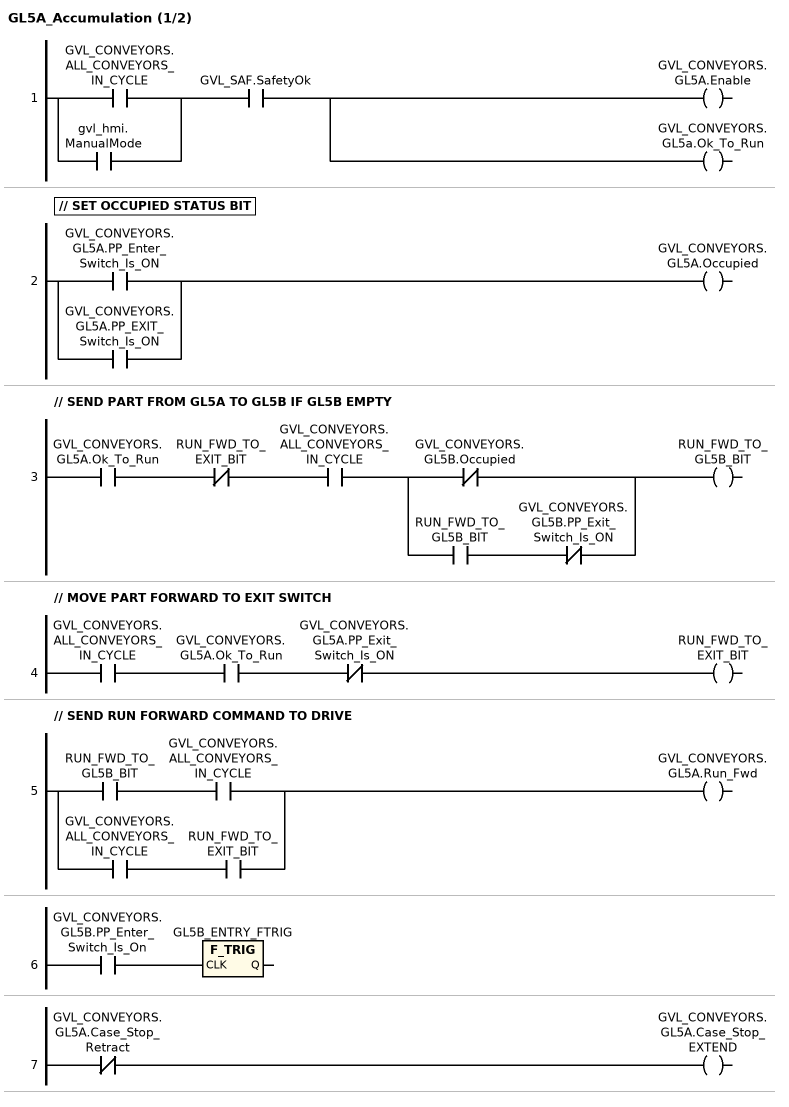
// NETWORK 1
_w1 := (GVL_CONVEYORS.ALL_CONVEYORS_IN_CYCLE OR gvl_hmi.ManualMode) AND GVL_SAF.SafetyOk;
GVL_CONVEYORS.GL5A.Enable := _w1;
GVL_CONVEYORS.GL5a.Ok_To_Run := _w1;

// NETWORK 2
// label: // SET OCCUPIED STATUS BIT
GVL_CONVEYORS.GL5A.Occupied := GVL_CONVEYORS.GL5A.PP_Enter_Switch_Is_ON OR GVL_CONVEYORS.GL5A.PP_EXIT_Switch_Is_ON;

// NETWORK 3: // SEND PART FROM GL5A TO GL5B IF GL5B EMPTY
RUN_FWD_TO_GL5B_BIT := GVL_CONVEYORS.GL5A.Ok_To_Run AND NOT RUN_FWD_TO_EXIT_BIT AND GVL_CONVEYORS.ALL_CONVEYORS_IN_CYCLE AND (NOT GVL_CONVEYORS.GL5B.Occupied OR RUN_FWD_TO_GL5B_BIT AND NOT GVL_CONVEYORS.GL5B.PP_Exit_Switch_Is_ON);

// NETWORK 4: // MOVE PART FORWARD TO EXIT SWITCH
RUN_FWD_TO_EXIT_BIT := GVL_CONVEYORS.ALL_CONVEYORS_IN_CYCLE AND GVL_CONVEYORS.GL5A.Ok_To_Run AND NOT GVL_CONVEYORS.GL5A.PP_Exit_Switch_Is_ON;

// NETWORK 5: // SEND RUN FORWARD COMMAND TO DRIVE
GVL_CONVEYORS.GL5A.Run_Fwd := RUN_FWD_TO_GL5B_BIT AND GVL_CONVEYORS.ALL_CONVEYORS_IN_CYCLE OR GVL_CONVEYORS.ALL_CONVEYORS_IN_CYCLE AND RUN_FWD_TO_EXIT_BIT;

// NETWORK 6
GL5B_ENTRY_FTRIG(CLK := GVL_CONVEYORS.GL5B.PP_Enter_Switch_Is_On); // F_TRIG

// NETWORK 7
GVL_CONVEYORS.GL5A.Case_Stop_EXTEND := NOT GVL_CONVEYORS.GL5A.Case_Stop_Retract;

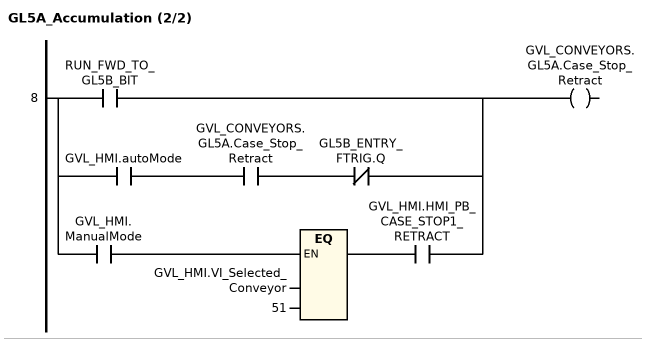
// NETWORK 8
GVL_CONVEYORS.GL5A.Case_Stop_Retract := RUN_FWD_TO_GL5B_BIT OR GVL_HMI.autoMode AND GVL_CONVEYORS.GL5A.Case_Stop_Retract AND NOT GL5B_ENTRY_FTRIG.Q OR (GVL_HMI.ManualMode AND GVL_HMI.VI_Selected_Conveyor = 51) AND GVL_HMI.HMI_PB_CASE_STOP1_RETRACT;

END_PROGRAM

// ---- Machine System/PRGs/Conveyors/GL5B_Accumulation.TcPOU
PROGRAM GL5B_Accumulation
VAR
	
	RUN_FWD_TO_GL2_BIT : BOOL; // GL2 EMPTY SO SEND PART FROM GL5B TO GL2
	RUN_FWD_TO_EXIT_BIT : BOOL; // RUN GL5B FWD TO EXIT SENSOR
	
END_VAR
VAR // added by the converter: edge detectors and wires of the graphical bodies
    _w1 : BOOL;
END_VAR

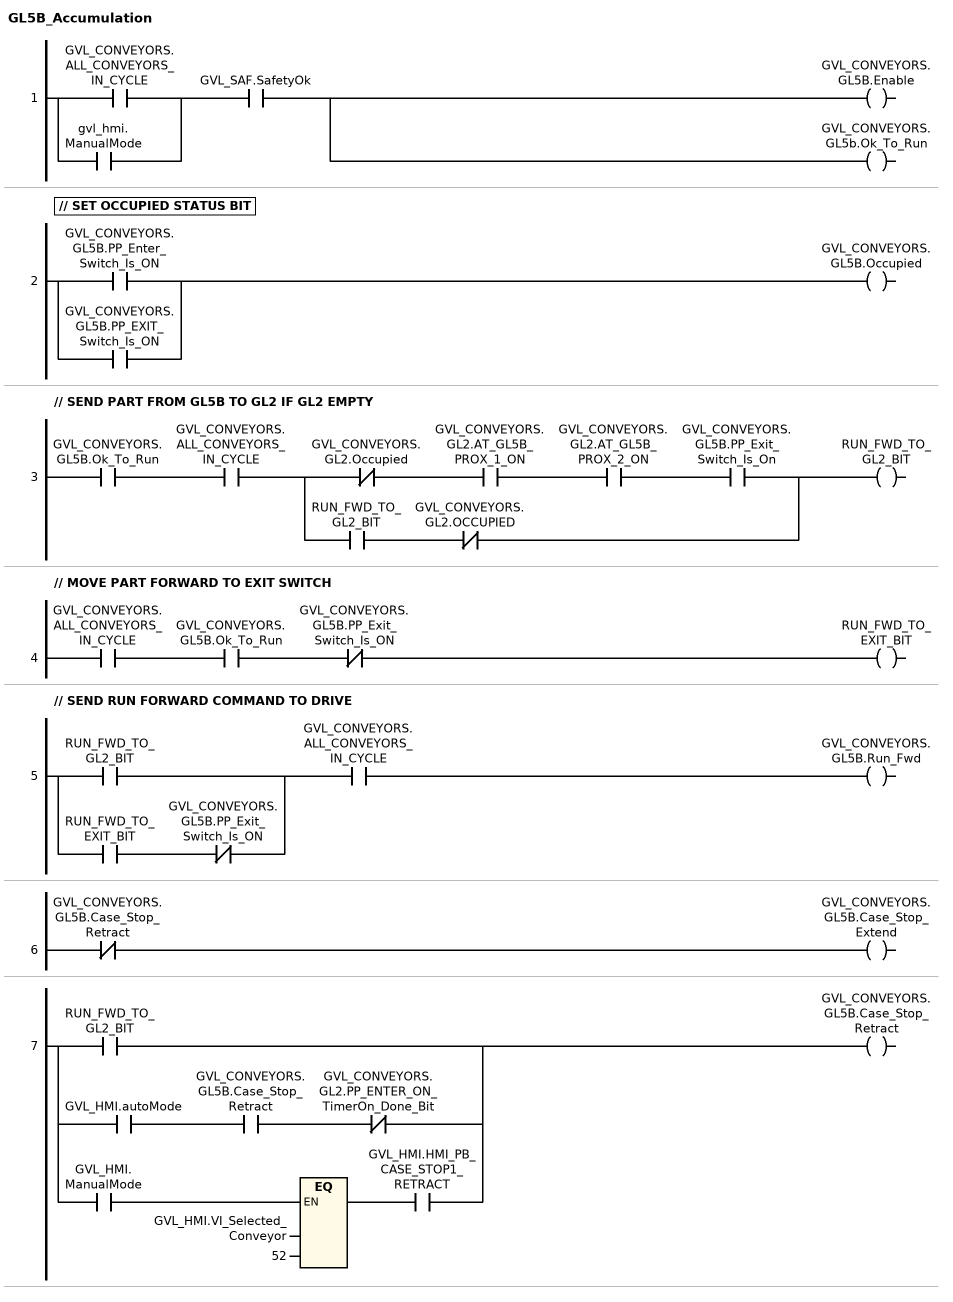
// NETWORK 1
_w1 := (GVL_CONVEYORS.ALL_CONVEYORS_IN_CYCLE OR gvl_hmi.ManualMode) AND GVL_SAF.SafetyOk;
GVL_CONVEYORS.GL5B.Enable := _w1;
GVL_CONVEYORS.GL5b.Ok_To_Run := _w1;

// NETWORK 2
// label: // SET OCCUPIED STATUS BIT
GVL_CONVEYORS.GL5B.Occupied := GVL_CONVEYORS.GL5B.PP_Enter_Switch_Is_ON OR GVL_CONVEYORS.GL5B.PP_EXIT_Switch_Is_ON;

// NETWORK 3: // SEND PART FROM GL5B TO GL2 IF GL2 EMPTY
RUN_FWD_TO_GL2_BIT := GVL_CONVEYORS.GL5B.Ok_To_Run AND GVL_CONVEYORS.ALL_CONVEYORS_IN_CYCLE AND (NOT GVL_CONVEYORS.GL2.Occupied AND GVL_CONVEYORS.GL2.AT_GL5B_PROX_1_ON AND GVL_CONVEYORS.GL2.AT_GL5B_PROX_2_ON AND GVL_CONVEYORS.GL5B.PP_Exit_Switch_Is_On OR RUN_FWD_TO_GL2_BIT AND NOT GVL_CONVEYORS.GL2.OCCUPIED);

// NETWORK 4: // MOVE PART FORWARD TO EXIT SWITCH
RUN_FWD_TO_EXIT_BIT := GVL_CONVEYORS.ALL_CONVEYORS_IN_CYCLE AND GVL_CONVEYORS.GL5B.Ok_To_Run AND NOT GVL_CONVEYORS.GL5B.PP_Exit_Switch_Is_ON;

// NETWORK 5: // SEND RUN FORWARD COMMAND TO DRIVE
GVL_CONVEYORS.GL5B.Run_Fwd := (RUN_FWD_TO_GL2_BIT OR RUN_FWD_TO_EXIT_BIT AND NOT GVL_CONVEYORS.GL5B.PP_Exit_Switch_Is_ON) AND GVL_CONVEYORS.ALL_CONVEYORS_IN_CYCLE;

// NETWORK 6
GVL_CONVEYORS.GL5B.Case_Stop_Extend := NOT GVL_CONVEYORS.GL5B.Case_Stop_Retract;

// NETWORK 7
GVL_CONVEYORS.GL5B.Case_Stop_Retract := RUN_FWD_TO_GL2_BIT OR GVL_HMI.autoMode AND GVL_CONVEYORS.GL5B.Case_Stop_Retract AND NOT GVL_CONVEYORS.GL2.PP_ENTER_ON_TimerOn_Done_Bit OR (GVL_HMI.ManualMode AND GVL_HMI.VI_Selected_Conveyor = 52) AND GVL_HMI.HMI_PB_CASE_STOP1_RETRACT;

END_PROGRAM

// ---- Machine System/PRGs/Conveyors/GL6_Conveyor.TcPOU
PROGRAM GL6_Conveyor
VAR
	GL6_RD: SRoll_Door;
	PASSSED_ROLL_DOOR : BOOL;
	RUN_FWD_BIT_TO_LOAD: BOOL; // RUN FORWARD TO LOAD POSITIONS
	RUN_FWD_BIT_TO_EXIT : BOOL; // RUN FORWARD TO EXIT POSITION AFTER DROP
	JoeBit : BOOL := FALSE;
END_VAR
VAR // added by the converter: edge detectors and wires of the graphical bodies
    _w1 : BOOL;
END_VAR

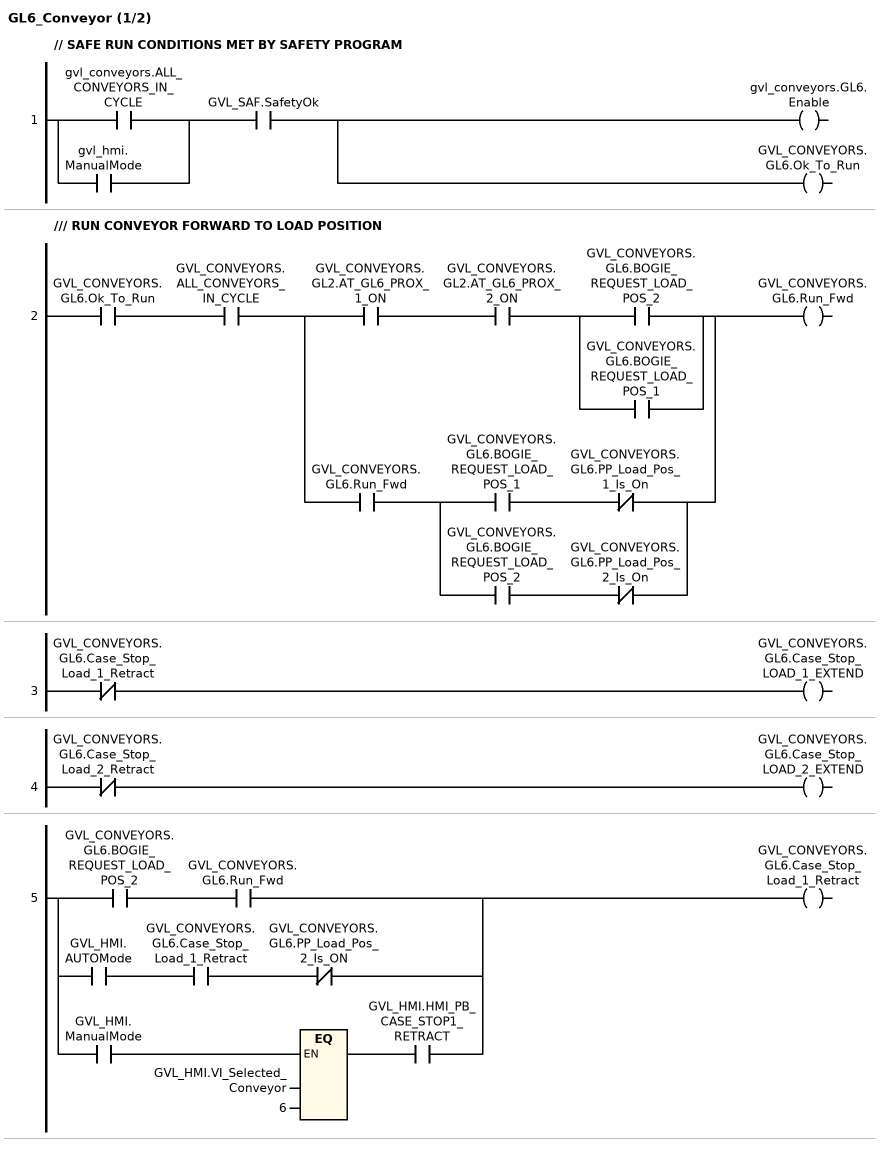
// NETWORK 1: // SAFE RUN CONDITIONS MET BY SAFETY PROGRAM
_w1 := (gvl_conveyors.ALL_CONVEYORS_IN_CYCLE OR gvl_hmi.ManualMode) AND GVL_SAF.SafetyOk;
gvl_conveyors.GL6.Enable := _w1;
GVL_CONVEYORS.GL6.Ok_To_Run := _w1;

// NETWORK 2: /// RUN CONVEYOR FORWARD TO LOAD POSITION
GVL_CONVEYORS.GL6.Run_Fwd := GVL_CONVEYORS.GL6.Ok_To_Run AND GVL_CONVEYORS.ALL_CONVEYORS_IN_CYCLE AND (GVL_CONVEYORS.GL2.AT_GL6_PROX_1_ON AND GVL_CONVEYORS.GL2.AT_GL6_PROX_2_ON AND (GVL_CONVEYORS.GL6.BOGIE_REQUEST_LOAD_POS_2 OR GVL_CONVEYORS.GL6.BOGIE_REQUEST_LOAD_POS_1) OR GVL_CONVEYORS.GL6.Run_Fwd AND (GVL_CONVEYORS.GL6.BOGIE_REQUEST_LOAD_POS_1 AND NOT GVL_CONVEYORS.GL6.PP_Load_Pos_1_Is_On OR GVL_CONVEYORS.GL6.BOGIE_REQUEST_LOAD_POS_2 AND NOT GVL_CONVEYORS.GL6.PP_Load_Pos_2_Is_On));

// NETWORK 3
GVL_CONVEYORS.GL6.Case_Stop_LOAD_1_EXTEND := NOT GVL_CONVEYORS.GL6.Case_Stop_Load_1_Retract;

// NETWORK 4
GVL_CONVEYORS.GL6.Case_Stop_LOAD_2_EXTEND := NOT GVL_CONVEYORS.GL6.Case_Stop_Load_2_Retract;

// NETWORK 5
GVL_CONVEYORS.GL6.Case_Stop_Load_1_Retract := GVL_CONVEYORS.GL6.BOGIE_REQUEST_LOAD_POS_2 AND GVL_CONVEYORS.GL6.Run_Fwd OR GVL_HMI.AUTOMode AND GVL_CONVEYORS.GL6.Case_Stop_Load_1_Retract AND NOT GVL_CONVEYORS.GL6.PP_Load_Pos_2_Is_ON OR (GVL_HMI.ManualMode AND GVL_HMI.VI_Selected_Conveyor = 6) AND GVL_HMI.HMI_PB_CASE_STOP1_RETRACT;

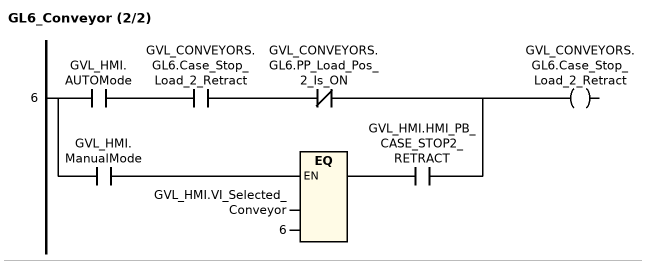
// NETWORK 6
GVL_CONVEYORS.GL6.Case_Stop_Load_2_Retract := GVL_HMI.AUTOMode AND GVL_CONVEYORS.GL6.Case_Stop_Load_2_Retract AND NOT GVL_CONVEYORS.GL6.PP_Load_Pos_2_Is_ON OR (GVL_HMI.ManualMode AND GVL_HMI.VI_Selected_Conveyor = 6) AND GVL_HMI.HMI_PB_CASE_STOP2_RETRACT;

END_PROGRAM

// ---- Machine System/PRGs/Conveyors/GL7_Conveyor.TcPOU
PROGRAM GL7_Conveyor
VAR
	
	RUN_FWD_BIT_TO_EXIT : BOOL; // RUN FORWARD TO EXIT POSITION AFTER DROP
END_VAR
VAR // added by the converter: edge detectors and wires of the graphical bodies
    _w1 : BOOL;
END_VAR

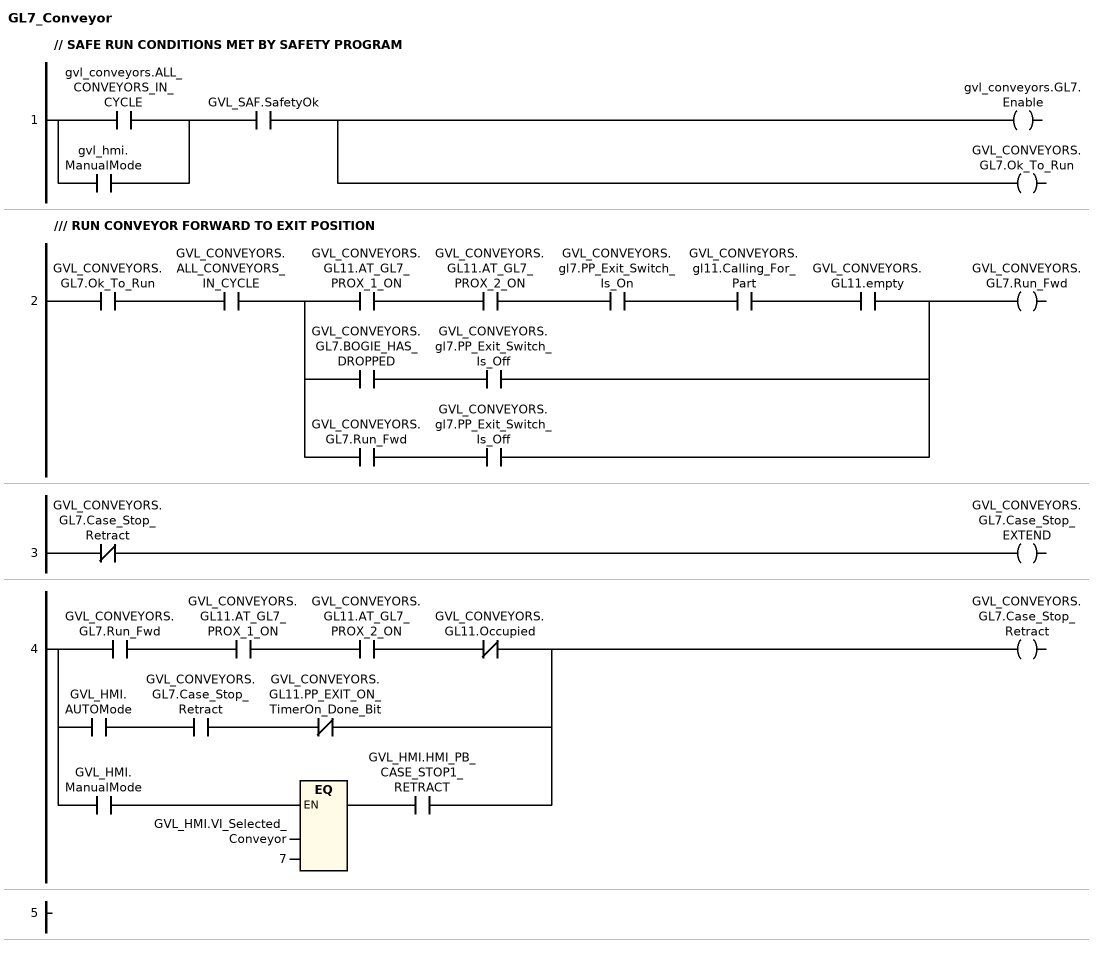
// NETWORK 1: // SAFE RUN CONDITIONS MET BY SAFETY PROGRAM
_w1 := (gvl_conveyors.ALL_CONVEYORS_IN_CYCLE OR gvl_hmi.ManualMode) AND GVL_SAF.SafetyOk;
gvl_conveyors.GL7.Enable := _w1;
GVL_CONVEYORS.GL7.Ok_To_Run := _w1;

// NETWORK 2: /// RUN CONVEYOR FORWARD TO EXIT POSITION
GVL_CONVEYORS.GL7.Run_Fwd := GVL_CONVEYORS.GL7.Ok_To_Run AND GVL_CONVEYORS.ALL_CONVEYORS_IN_CYCLE AND (GVL_CONVEYORS.GL11.AT_GL7_PROX_1_ON AND GVL_CONVEYORS.GL11.AT_GL7_PROX_2_ON AND GVL_CONVEYORS.gl7.PP_Exit_Switch_Is_On AND GVL_CONVEYORS.gl11.Calling_For_Part AND GVL_CONVEYORS.GL11.empty OR GVL_CONVEYORS.GL7.BOGIE_HAS_DROPPED AND GVL_CONVEYORS.gl7.PP_Exit_Switch_Is_Off OR GVL_CONVEYORS.GL7.Run_Fwd AND GVL_CONVEYORS.gl7.PP_Exit_Switch_Is_Off);

// NETWORK 3
GVL_CONVEYORS.GL7.Case_Stop_EXTEND := NOT GVL_CONVEYORS.GL7.Case_Stop_Retract;

// NETWORK 4
GVL_CONVEYORS.GL7.Case_Stop_Retract := GVL_CONVEYORS.GL7.Run_Fwd AND GVL_CONVEYORS.GL11.AT_GL7_PROX_1_ON AND GVL_CONVEYORS.GL11.AT_GL7_PROX_2_ON AND NOT GVL_CONVEYORS.GL11.Occupied OR GVL_HMI.AUTOMode AND GVL_CONVEYORS.GL7.Case_Stop_Retract AND NOT GVL_CONVEYORS.GL11.PP_EXIT_ON_TimerOn_Done_Bit OR (GVL_HMI.ManualMode AND GVL_HMI.VI_Selected_Conveyor = 7) AND GVL_HMI.HMI_PB_CASE_STOP1_RETRACT;

// NETWORK 5

END_PROGRAM

// ---- Machine System/PRGs/Conveyors/GL8_Conveyor.TcPOU
PROGRAM GL8_Conveyor
VAR
	
	GL8_RD: SRoll_Door;
	PASSSED_ROLL_DOOR : BOOL;
	RUN_FWD_BIT_TO_LOAD: BOOL; // RUN FORWARD TO LOAD POSITIONS
	RUN_FWD_BIT_TO_EXIT : BOOL; // RUN FORWARD TO EXIT POSITION AFTER DROP
	
END_VAR
VAR // added by the converter: edge detectors and wires of the graphical bodies
    _w1 : BOOL;
END_VAR

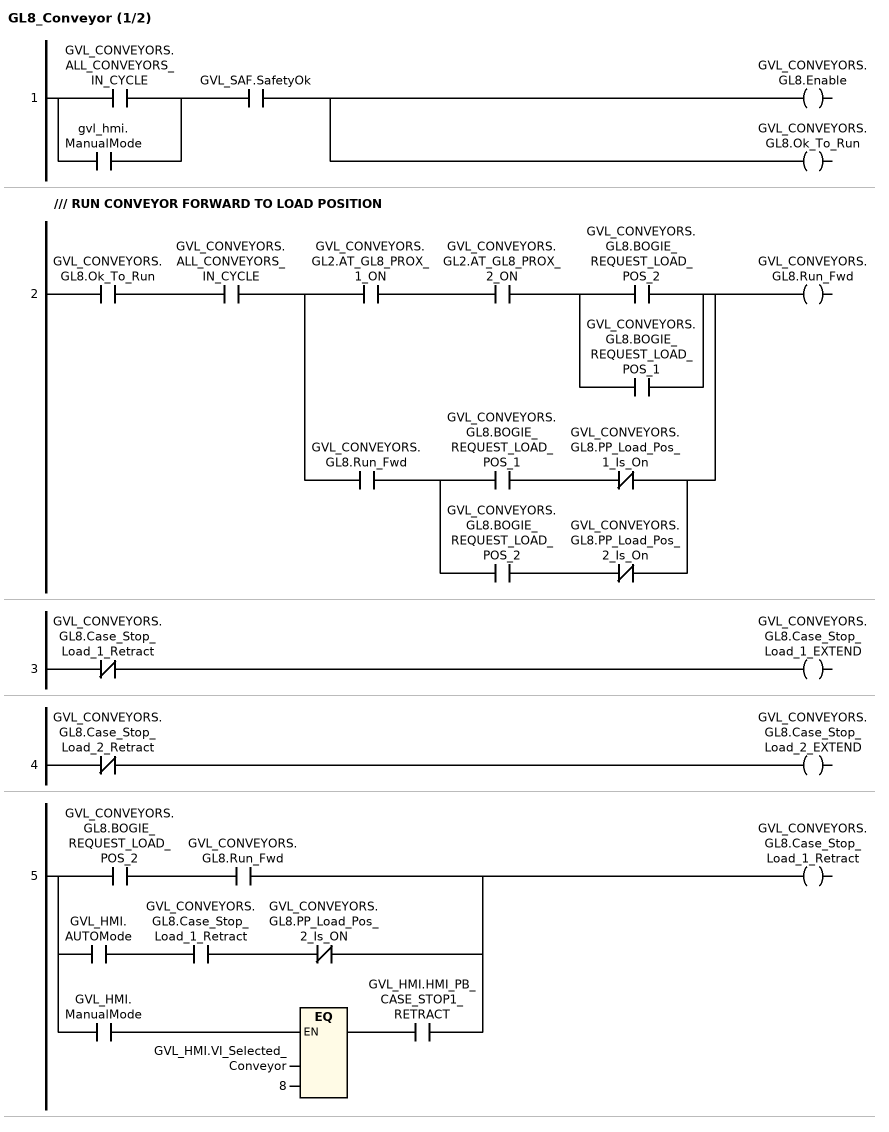
// NETWORK 1
_w1 := (GVL_CONVEYORS.ALL_CONVEYORS_IN_CYCLE OR gvl_hmi.ManualMode) AND GVL_SAF.SafetyOk;
GVL_CONVEYORS.GL8.Enable := _w1;
GVL_CONVEYORS.GL8.Ok_To_Run := _w1;

// NETWORK 2: /// RUN CONVEYOR FORWARD TO LOAD POSITION
GVL_CONVEYORS.GL8.Run_Fwd := GVL_CONVEYORS.GL8.Ok_To_Run AND GVL_CONVEYORS.ALL_CONVEYORS_IN_CYCLE AND (GVL_CONVEYORS.GL2.AT_GL8_PROX_1_ON AND GVL_CONVEYORS.GL2.AT_GL8_PROX_2_ON AND (GVL_CONVEYORS.GL8.BOGIE_REQUEST_LOAD_POS_2 OR GVL_CONVEYORS.GL8.BOGIE_REQUEST_LOAD_POS_1) OR GVL_CONVEYORS.GL8.Run_Fwd AND (GVL_CONVEYORS.GL8.BOGIE_REQUEST_LOAD_POS_1 AND NOT GVL_CONVEYORS.GL8.PP_Load_Pos_1_Is_On OR GVL_CONVEYORS.GL8.BOGIE_REQUEST_LOAD_POS_2 AND NOT GVL_CONVEYORS.GL8.PP_Load_Pos_2_Is_On));

// NETWORK 3
GVL_CONVEYORS.GL8.Case_Stop_Load_1_EXTEND := NOT GVL_CONVEYORS.GL8.Case_Stop_Load_1_Retract;

// NETWORK 4
GVL_CONVEYORS.GL8.Case_Stop_Load_2_EXTEND := NOT GVL_CONVEYORS.GL8.Case_Stop_Load_2_Retract;

// NETWORK 5
GVL_CONVEYORS.GL8.Case_Stop_Load_1_Retract := GVL_CONVEYORS.GL8.BOGIE_REQUEST_LOAD_POS_2 AND GVL_CONVEYORS.GL8.Run_Fwd OR GVL_HMI.AUTOMode AND GVL_CONVEYORS.GL8.Case_Stop_Load_1_Retract AND NOT GVL_CONVEYORS.GL8.PP_Load_Pos_2_Is_ON OR (GVL_HMI.ManualMode AND GVL_HMI.VI_Selected_Conveyor = 8) AND GVL_HMI.HMI_PB_CASE_STOP1_RETRACT;

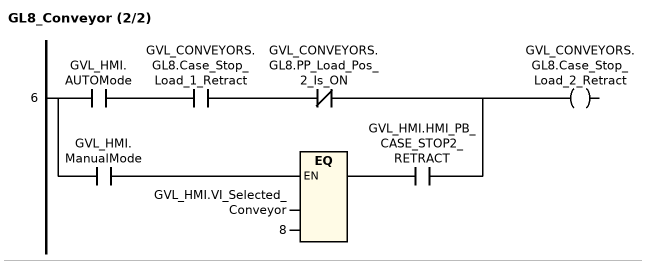
// NETWORK 6
GVL_CONVEYORS.GL8.Case_Stop_Load_2_Retract := GVL_HMI.AUTOMode AND GVL_CONVEYORS.GL8.Case_Stop_Load_1_Retract AND NOT GVL_CONVEYORS.GL8.PP_Load_Pos_2_Is_ON OR (GVL_HMI.ManualMode AND GVL_HMI.VI_Selected_Conveyor = 8) AND GVL_HMI.HMI_PB_CASE_STOP2_RETRACT;

END_PROGRAM

// ---- Machine System/PRGs/Conveyors/GL9_Conveyor.TcPOU
PROGRAM GL9_Conveyor
VAR
	
	RUN_FWD_BIT_TO_EXIT : BOOL; // RUN FORWARD TO EXIT POSITION AFTER DROP
END_VAR
VAR // added by the converter: edge detectors and wires of the graphical bodies
    _w1 : BOOL;
END_VAR

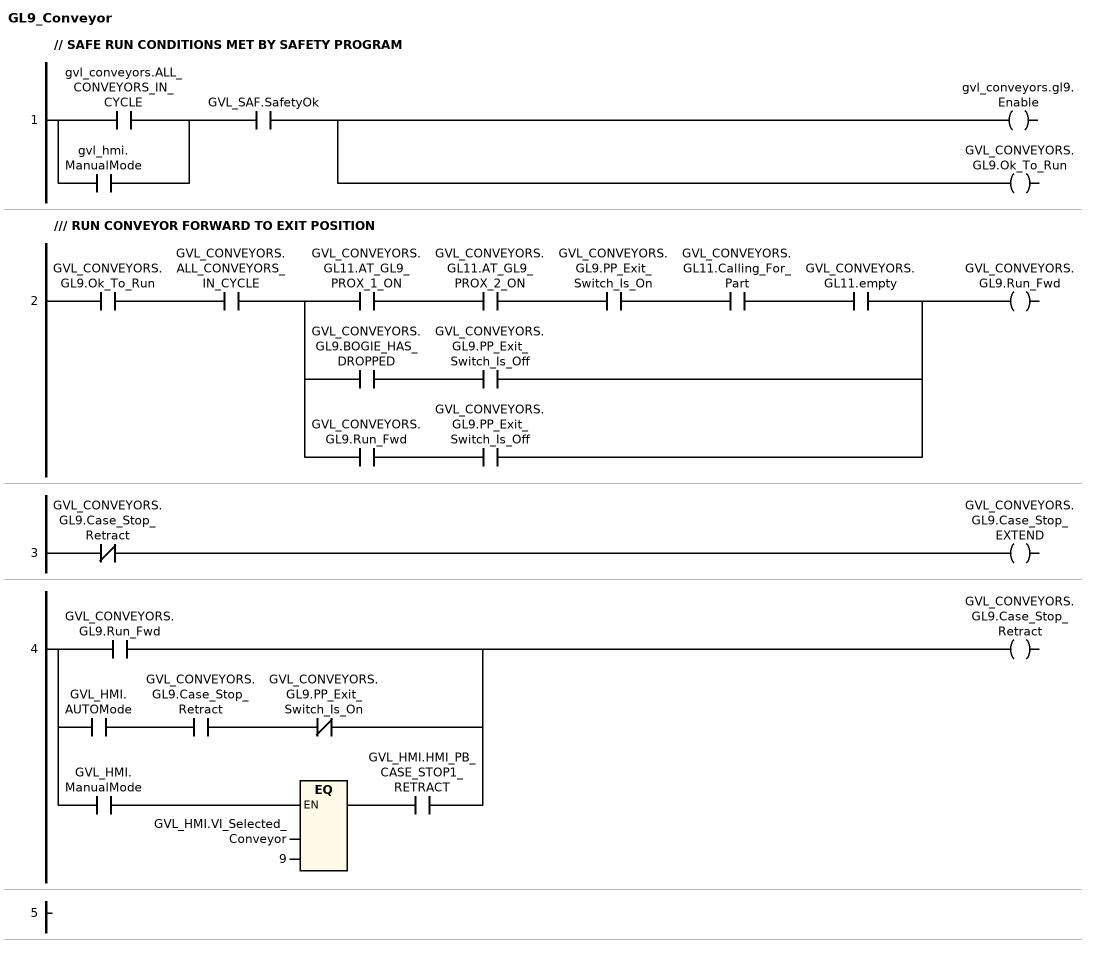
// NETWORK 1: // SAFE RUN CONDITIONS MET BY SAFETY PROGRAM
_w1 := (gvl_conveyors.ALL_CONVEYORS_IN_CYCLE OR gvl_hmi.ManualMode) AND GVL_SAF.SafetyOk;
gvl_conveyors.gl9.Enable := _w1;
GVL_CONVEYORS.GL9.Ok_To_Run := _w1;

// NETWORK 2: /// RUN CONVEYOR FORWARD TO EXIT POSITION
GVL_CONVEYORS.GL9.Run_Fwd := GVL_CONVEYORS.GL9.Ok_To_Run AND GVL_CONVEYORS.ALL_CONVEYORS_IN_CYCLE AND (GVL_CONVEYORS.GL11.AT_GL9_PROX_1_ON AND GVL_CONVEYORS.GL11.AT_GL9_PROX_2_ON AND GVL_CONVEYORS.GL9.PP_Exit_Switch_Is_On AND GVL_CONVEYORS.GL11.Calling_For_Part AND GVL_CONVEYORS.GL11.empty OR GVL_CONVEYORS.GL9.BOGIE_HAS_DROPPED AND GVL_CONVEYORS.GL9.PP_Exit_Switch_Is_Off OR GVL_CONVEYORS.GL9.Run_Fwd AND GVL_CONVEYORS.GL9.PP_Exit_Switch_Is_Off);

// NETWORK 3
GVL_CONVEYORS.GL9.Case_Stop_EXTEND := NOT GVL_CONVEYORS.GL9.Case_Stop_Retract;

// NETWORK 4
GVL_CONVEYORS.GL9.Case_Stop_Retract := GVL_CONVEYORS.GL9.Run_Fwd OR GVL_HMI.AUTOMode AND GVL_CONVEYORS.GL9.Case_Stop_Retract AND NOT GVL_CONVEYORS.GL9.PP_Exit_Switch_Is_On OR (GVL_HMI.ManualMode AND GVL_HMI.VI_Selected_Conveyor = 9) AND GVL_HMI.HMI_PB_CASE_STOP1_RETRACT;

// NETWORK 5

END_PROGRAM

// ---- Machine System/PRGs/Rib Machine/Guarding_Safety.TcPOU
PROGRAM Guarding_Safety
VAR
END_VAR

// NETWORK 1

END_PROGRAM

// ---- Machine System/PRGs/Rib Machine/Input_Buffering_RB.TcPOU
PROGRAM Input_Buffering_RB
VAR PERSISTENT
	
	StackerPartPresentTon: TON;
	StackerPinExtendedTon: TON;
	StackerPinRetractedTon: TON;
	IndexerPartPresentTon: TON;
    SawExtendedTon: TON;
	SawRetractedTon: TON;
	SawClampExtendedTon: TON;
	SawClampRetractedTon: TON;
	SawClampOpenTon: TON;
	SawClampClosedTon: TON;
	TransferClampOpenTon: TON;
	TransferClampClosedTon: TON;
	TransferClampExtdTon: TON;
	TransferClampRetdTon: TON;
	TransferExtdTon: TON;
	TransferRetdTon: TON;
	RibHoistUpTon: TON;
	RibHoistDownTon: TON;
	EjectExtendedTon: TON;
	EjectRetractedTon: TON;
	AirPressureSwitchTon: TON;
	IndexerHomeTon: TON;
	
END_VAR

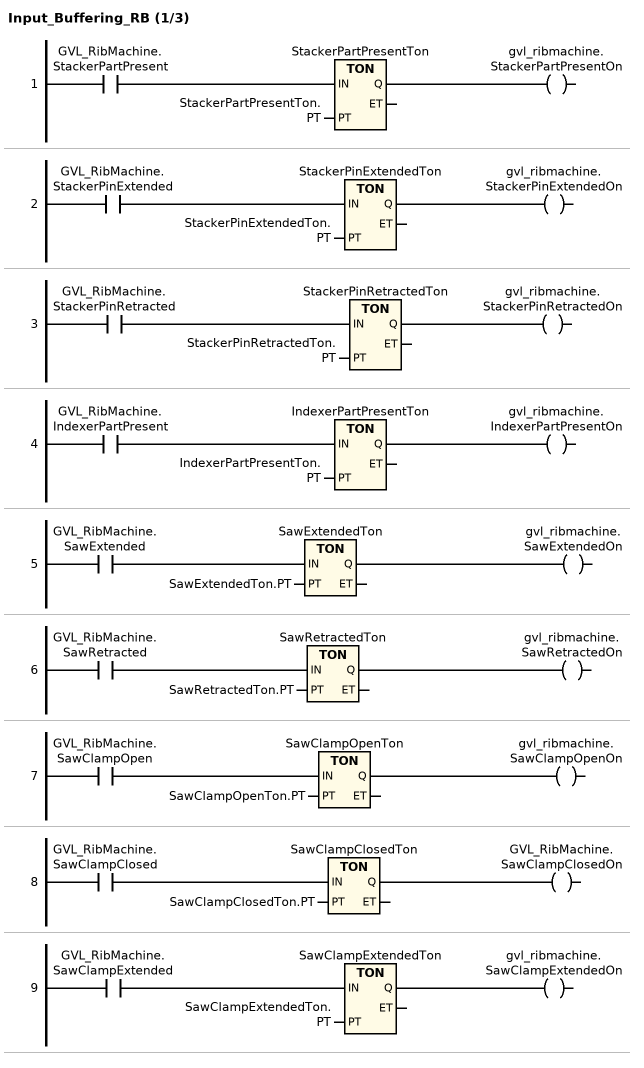
// NETWORK 1
StackerPartPresentTon(IN := GVL_RibMachine.StackerPartPresent, PT := StackerPartPresentTon.PT); // TON
gvl_ribmachine.StackerPartPresentOn := StackerPartPresentTon.Q;

// NETWORK 2
StackerPinExtendedTon(IN := GVL_RibMachine.StackerPinExtended, PT := StackerPinExtendedTon.PT); // TON
gvl_ribmachine.StackerPinExtendedOn := StackerPinExtendedTon.Q;

// NETWORK 3
StackerPinRetractedTon(IN := GVL_RibMachine.StackerPinRetracted, PT := StackerPinRetractedTon.PT); // TON
gvl_ribmachine.StackerPinRetractedOn := StackerPinRetractedTon.Q;

// NETWORK 4
IndexerPartPresentTon(IN := GVL_RibMachine.IndexerPartPresent, PT := IndexerPartPresentTon.PT); // TON
gvl_ribmachine.IndexerPartPresentOn := IndexerPartPresentTon.Q;

// NETWORK 5
SawExtendedTon(IN := GVL_RibMachine.SawExtended, PT := SawExtendedTon.PT); // TON
gvl_ribmachine.SawExtendedOn := SawExtendedTon.Q;

// NETWORK 6
SawRetractedTon(IN := GVL_RibMachine.SawRetracted, PT := SawRetractedTon.PT); // TON
gvl_ribmachine.SawRetractedOn := SawRetractedTon.Q;

// NETWORK 7
SawClampOpenTon(IN := GVL_RibMachine.SawClampOpen, PT := SawClampOpenTon.PT); // TON
gvl_ribmachine.SawClampOpenOn := SawClampOpenTon.Q;

// NETWORK 8
SawClampClosedTon(IN := GVL_RibMachine.SawClampClosed, PT := SawClampClosedTon.PT); // TON
GVL_RibMachine.SawClampClosedOn := SawClampClosedTon.Q;

// NETWORK 9
SawClampExtendedTon(IN := GVL_RibMachine.SawClampExtended, PT := SawClampExtendedTon.PT); // TON
gvl_ribmachine.SawClampExtendedOn := SawClampExtendedTon.Q;

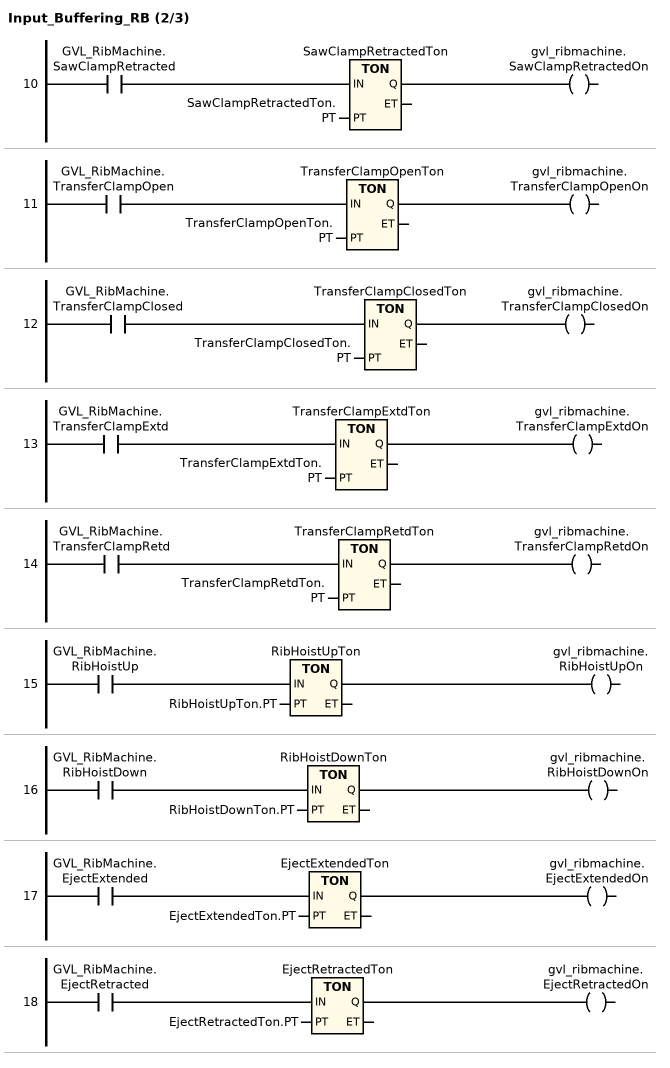
// NETWORK 10
SawClampRetractedTon(IN := GVL_RibMachine.SawClampRetracted, PT := SawClampRetractedTon.PT); // TON
gvl_ribmachine.SawClampRetractedOn := SawClampRetractedTon.Q;

// NETWORK 11
TransferClampOpenTon(IN := GVL_RibMachine.TransferClampOpen, PT := TransferClampOpenTon.PT); // TON
gvl_ribmachine.TransferClampOpenOn := TransferClampOpenTon.Q;

// NETWORK 12
TransferClampClosedTon(IN := GVL_RibMachine.TransferClampClosed, PT := TransferClampClosedTon.PT); // TON
gvl_ribmachine.TransferClampClosedOn := TransferClampClosedTon.Q;

// NETWORK 13
TransferClampExtdTon(IN := GVL_RibMachine.TransferClampExtd, PT := TransferClampExtdTon.PT); // TON
gvl_ribmachine.TransferClampExtdOn := TransferClampExtdTon.Q;

// NETWORK 14
TransferClampRetdTon(IN := GVL_RibMachine.TransferClampRetd, PT := TransferClampRetdTon.PT); // TON
gvl_ribmachine.TransferClampRetdOn := TransferClampRetdTon.Q;

// NETWORK 15
RibHoistUpTon(IN := GVL_RibMachine.RibHoistUp, PT := RibHoistUpTon.PT); // TON
gvl_ribmachine.RibHoistUpOn := RibHoistUpTon.Q;

// NETWORK 16
RibHoistDownTon(IN := GVL_RibMachine.RibHoistDown, PT := RibHoistDownTon.PT); // TON
gvl_ribmachine.RibHoistDownOn := RibHoistDownTon.Q;

// NETWORK 17
EjectExtendedTon(IN := GVL_RibMachine.EjectExtended, PT := EjectExtendedTon.PT); // TON
gvl_ribmachine.EjectExtendedOn := EjectExtendedTon.Q;

// NETWORK 18
EjectRetractedTon(IN := GVL_RibMachine.EjectRetracted, PT := EjectRetractedTon.PT); // TON
gvl_ribmachine.EjectRetractedOn := EjectRetractedTon.Q;

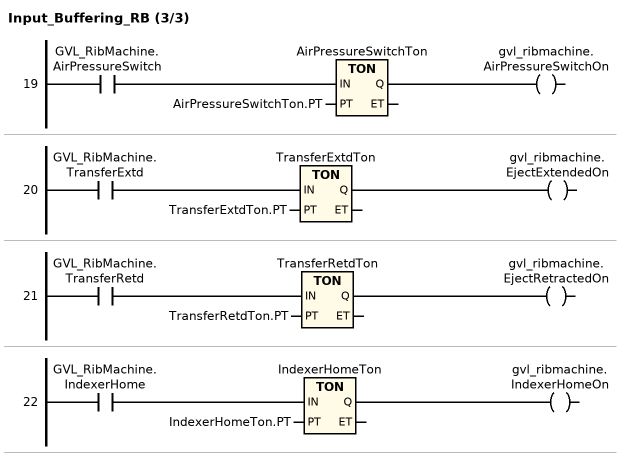
// NETWORK 19
AirPressureSwitchTon(IN := GVL_RibMachine.AirPressureSwitch, PT := AirPressureSwitchTon.PT); // TON
gvl_ribmachine.AirPressureSwitchOn := AirPressureSwitchTon.Q;

// NETWORK 20
TransferExtdTon(IN := GVL_RibMachine.TransferExtd, PT := TransferExtdTon.PT); // TON
gvl_ribmachine.EjectExtendedOn := TransferExtdTon.Q;

// NETWORK 21
TransferRetdTon(IN := GVL_RibMachine.TransferRetd, PT := TransferRetdTon.PT); // TON
gvl_ribmachine.EjectRetractedOn := TransferRetdTon.Q;

// NETWORK 22
IndexerHomeTon(IN := GVL_RibMachine.IndexerHome, PT := IndexerHomeTon.PT); // TON
gvl_ribmachine.IndexerHomeOn := IndexerHomeTon.Q;

END_PROGRAM

// ---- Machine System/PRGs/START_STOP.TcPOU
PROGRAM START_STOP
VAR
	START_TIMER : TON;
	START_TIMER_ELAPSED: TIME;
	START_TIMER_DONE : BOOL; 
	ALARM_HORN AT %Q* : BOOL; // CONVEYOR STARTING WARNING SIGNAL
	ALL_CONVEYORS_START_PB  AT %I*:  BOOL; // TIE THIS TO THE START COMMAND FROM HMI OR BUTTON
	ALL_CONVEYORS_STOP_PB  AT %I*: BOOL; // TIE THIS TO THE STOP COMMAND FROM HMI OR BUTTON
	START_PB_LT AT %Q*: BOOL; // START PB LIGHT
	STOP_PB_LT AT %Q*: BOOL; // STOP PB LIGHT
	KIRK_BIT: BOOL;
	HMI_CONVEYOR_START: BOOL; // START SIGNAL FROM HMI
	
END_VAR

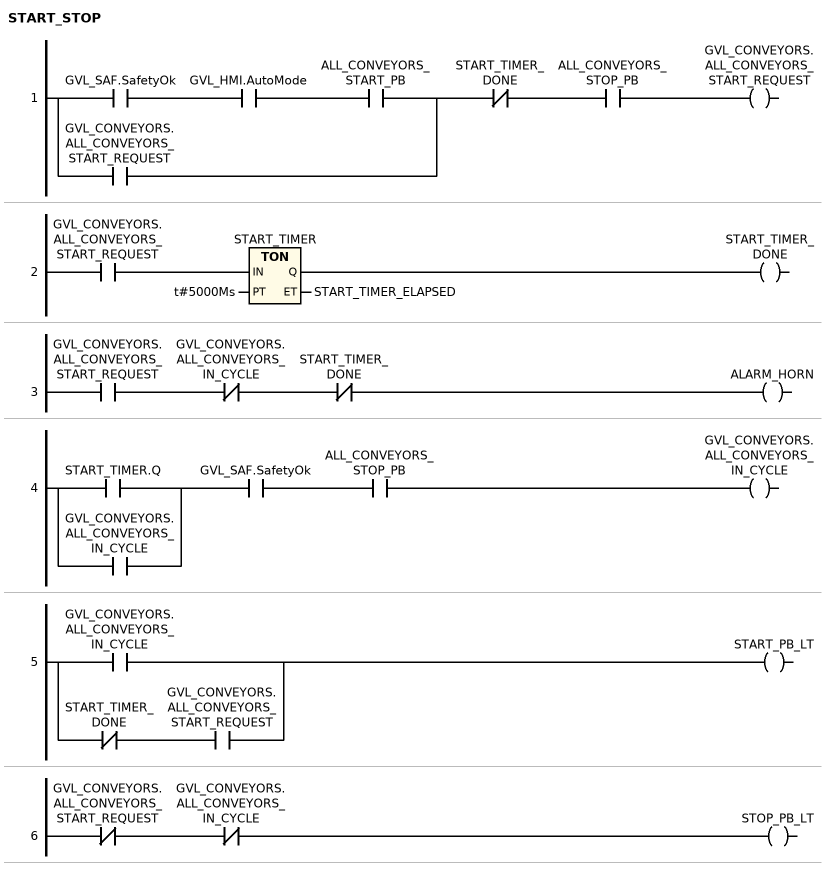
// NETWORK 1
GVL_CONVEYORS.ALL_CONVEYORS_START_REQUEST := (GVL_SAF.SafetyOk AND GVL_HMI.AutoMode AND ALL_CONVEYORS_START_PB OR GVL_CONVEYORS.ALL_CONVEYORS_START_REQUEST) AND NOT START_TIMER_DONE AND ALL_CONVEYORS_STOP_PB;

// NETWORK 2
START_TIMER(IN := GVL_CONVEYORS.ALL_CONVEYORS_START_REQUEST, PT := t#5000Ms, ET => START_TIMER_ELAPSED); // TON
START_TIMER_DONE := START_TIMER.Q;

// NETWORK 3
ALARM_HORN := GVL_CONVEYORS.ALL_CONVEYORS_START_REQUEST AND NOT GVL_CONVEYORS.ALL_CONVEYORS_IN_CYCLE AND NOT START_TIMER_DONE;

// NETWORK 4
GVL_CONVEYORS.ALL_CONVEYORS_IN_CYCLE := (START_TIMER.Q OR GVL_CONVEYORS.ALL_CONVEYORS_IN_CYCLE) AND GVL_SAF.SafetyOk AND ALL_CONVEYORS_STOP_PB;

// NETWORK 5
START_PB_LT := GVL_CONVEYORS.ALL_CONVEYORS_IN_CYCLE OR NOT START_TIMER_DONE AND GVL_CONVEYORS.ALL_CONVEYORS_START_REQUEST;

// NETWORK 6
STOP_PB_LT := NOT GVL_CONVEYORS.ALL_CONVEYORS_START_REQUEST AND NOT GVL_CONVEYORS.ALL_CONVEYORS_IN_CYCLE;

END_PROGRAM

// ---- Machine System/PRGs/Rib Machine/Index_and_Measure.TcPOU
PROGRAM Index_and_Measure
VAR
	RequestedRibLength:REAL; // Length in inches needed for ribs to cut
	MinRibLength: DINT; // Minimnm length of leftover that can still be used.
	MaxRibLength: DINT; // Longest rib lenght
	NumOfRibs:INT; // Quantity of tibs needed for next part
	RibRequest:BOOL; // Ribs needed for next part.
	RemainingLength:DINT; // Left over length of rib after cut
	PPI:REAL; // Pulses Per Inch from encoder
	CutLength: REAL; // Rib length to cut in encoder pulses 
	KerfWidth : REAL; // Width of saw blade in encoder pulses
	TotalCutLength : REAL; // Cut length requested plus kerf width of saw blade
	RibReadyToCut: BOOL; // Rib is in position to begin cutting
	HMI_PB_ManualJogFwd:BOOL; // HMI manual jog forward
	HMI_PB_ManualJogRev: bool; // HMI manual jog reverse
	IndexFwd: BOOL; // Clear path signal to go forward direction
	IndexRev: BOOL; // Clear path signal to go reverse direction
	OpenTransferClampRequest: BOOL;
	CloseTransferClampRequest: BOOL;
END_VAR

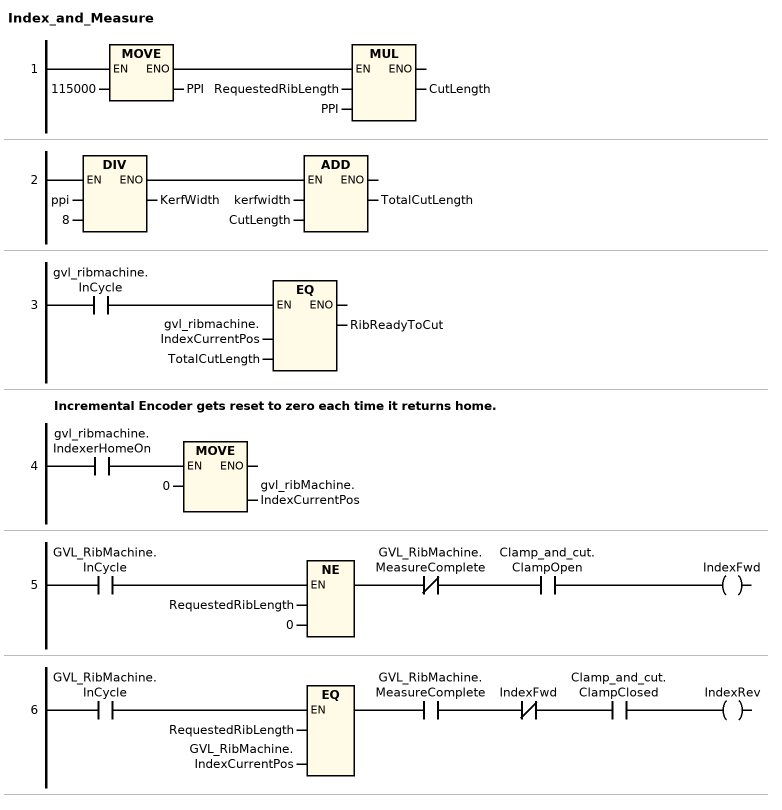
// NETWORK 1
PPI := 115000;
CutLength := RequestedRibLength * PPI;

// NETWORK 2
KerfWidth := ppi / 8;
TotalCutLength := kerfwidth + CutLength;

// NETWORK 3
IF gvl_ribmachine.InCycle THEN RibReadyToCut := gvl_ribmachine.IndexCurrentPos = TotalCutLength; END_IF

// NETWORK 4: Incremental Encoder gets reset to zero each time it returns home.
IF gvl_ribmachine.IndexerHomeOn THEN gvl_ribMachine.IndexCurrentPos := 0; END_IF

// NETWORK 5
IndexFwd := (GVL_RibMachine.InCycle AND RequestedRibLength <> 0) AND NOT GVL_RibMachine.MeasureComplete AND Clamp_and_cut.ClampOpen;

// NETWORK 6
IndexRev := (GVL_RibMachine.InCycle AND RequestedRibLength = GVL_RibMachine.IndexCurrentPos) AND GVL_RibMachine.MeasureComplete AND NOT IndexFwd AND Clamp_and_cut.ClampClosed;

END_PROGRAM

// ---- Machine System/PRGs/Rib Machine/Clamp_and_cut.TcPOU
PROGRAM Clamp_and_cut
VAR
	
	
	SawHome: BOOL; //Indexer is retracted to HOME switch
	SawTraversing: BOOL; // Saw is cycling through cutting
	SawDwellTimer: ton; // Dwell timer to wait for saw to spool up to speed
	SawExtended: BOOL; // Saw slide is fully extended
	ClampOpen: BOOL; // Saw clamp is open to receive part
	ClampClosed: BOOL; // Saw clamp is closed on to the part
	SawMotorRunning: BOOL; // Saw blade is spinning and motor not faulted
	CloseClampRequest: BOOL; // Logic bit to close saw clamp
	OpenClampRequest: BOOL; // Logic bit to open saw clamp
	SawDwellTimerElapsed: TIME; // Elapsed time of dwell timer
	SawDwellDoneBit: BOOL; // Dwell timer done bit
	StartSawRequest: BOOL; // Logic bit to start saw motor
	TraverseDwellTimer: ton; // Dwell timer to wait for traverse motor to spool up to speed
	TraverseDwellTimerElapsed: TIME; // Elapsed time of dwell timer
	TraverseDwellDoneBit: BOOL; // Dwell timer done bit
	DustCollectStartRequest: BOOL; // Logic bit to start dust collector
	
END_VAR
VAR // added by the converter: edge detectors and wires of the graphical bodies
    _rt1, _rt2, _rt3 : R_TRIG;
    _w1 : BOOL;
END_VAR

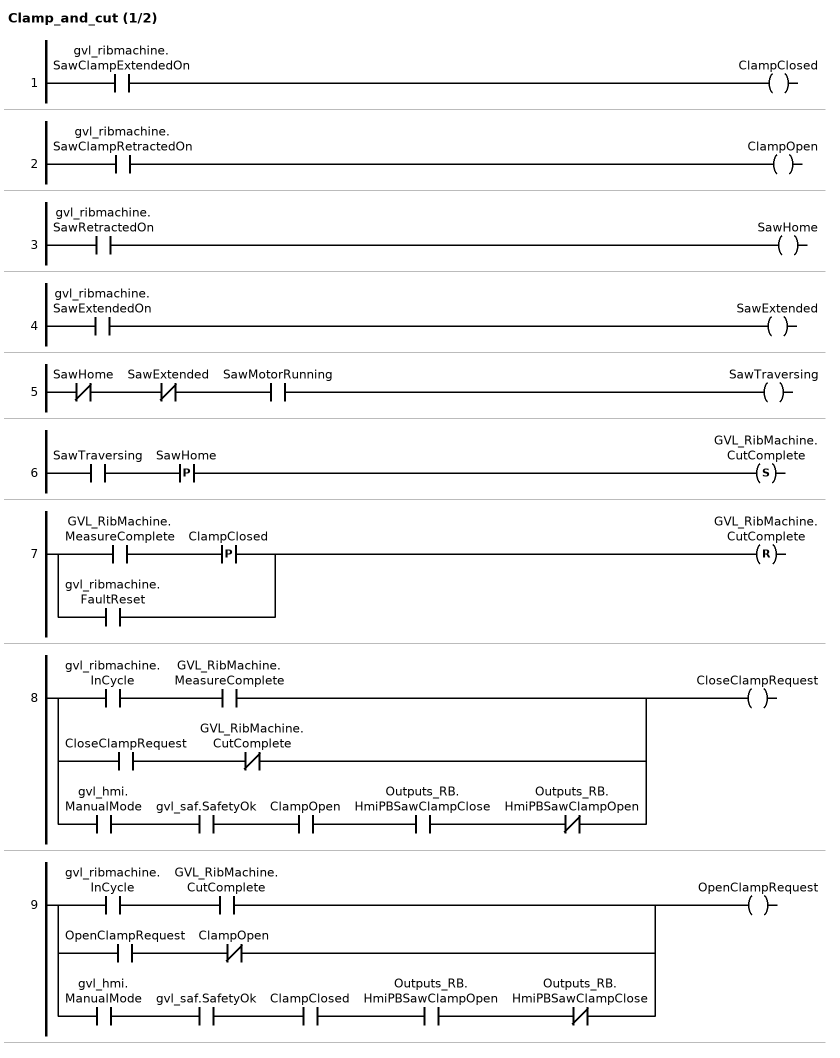
// NETWORK 1
ClampClosed := gvl_ribmachine.SawClampExtendedOn;

// NETWORK 2
ClampOpen := gvl_ribmachine.SawClampRetractedOn;

// NETWORK 3
SawHome := gvl_ribmachine.SawRetractedOn;

// NETWORK 4
SawExtended := gvl_ribmachine.SawExtendedOn;

// NETWORK 5
SawTraversing := NOT SawHome AND NOT SawExtended AND SawMotorRunning;

// NETWORK 6
_rt1(CLK := SawHome);
GVL_RibMachine.CutComplete S= SawTraversing AND _rt1.Q;

// NETWORK 7
_rt2(CLK := ClampClosed);
GVL_RibMachine.CutComplete R= GVL_RibMachine.MeasureComplete AND _rt2.Q OR gvl_ribmachine.FaultReset;

// NETWORK 8
CloseClampRequest := gvl_ribmachine.InCycle AND GVL_RibMachine.MeasureComplete OR CloseClampRequest AND NOT GVL_RibMachine.CutComplete OR gvl_hmi.ManualMode AND gvl_saf.SafetyOk AND ClampOpen AND Outputs_RB.HmiPBSawClampClose AND NOT Outputs_RB.HmiPBSawClampOpen;

// NETWORK 9
OpenClampRequest := gvl_ribmachine.InCycle AND GVL_RibMachine.CutComplete OR OpenClampRequest AND NOT ClampOpen OR gvl_hmi.ManualMode AND gvl_saf.SafetyOk AND ClampClosed AND Outputs_RB.HmiPBSawClampOpen AND NOT Outputs_RB.HmiPBSawClampClose;

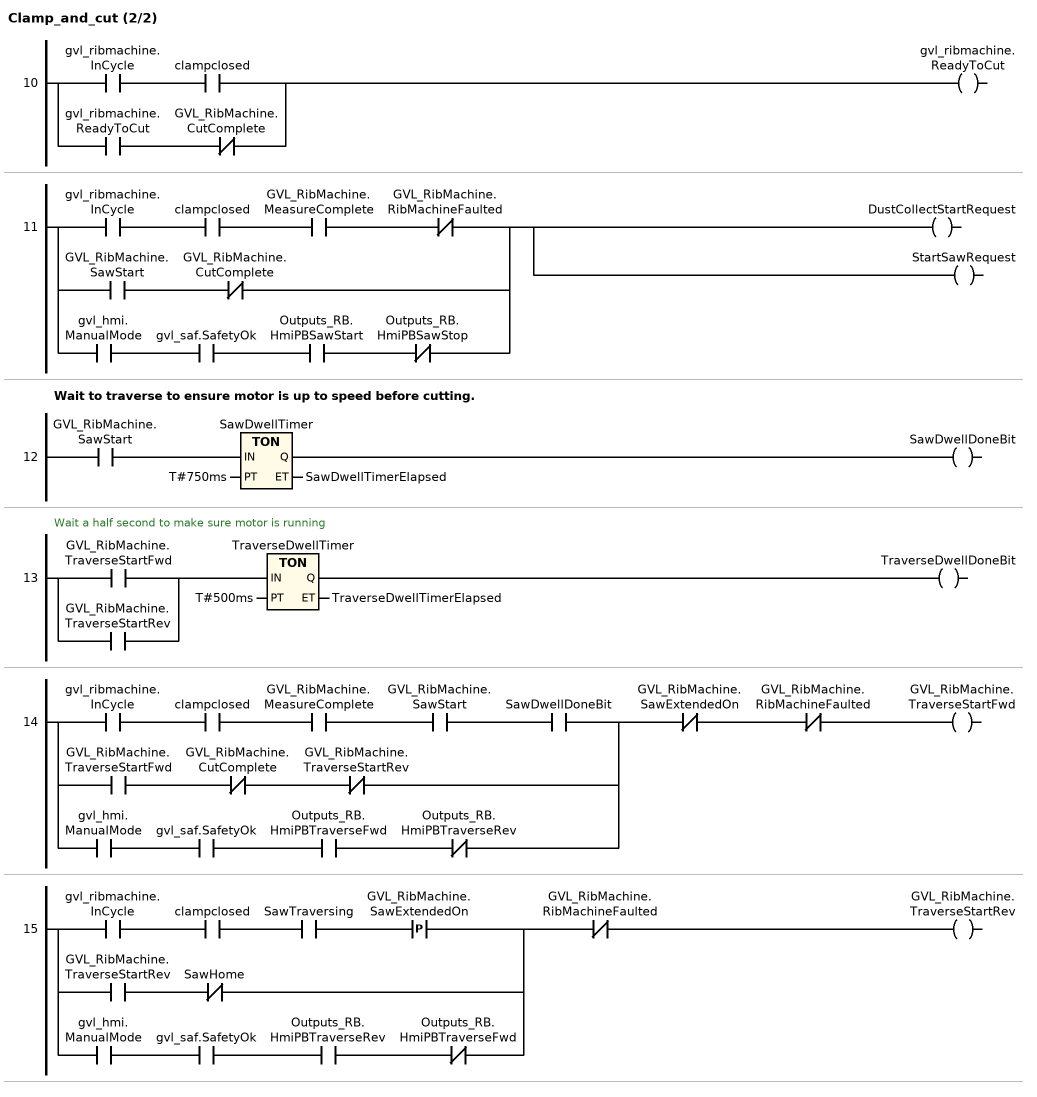
// NETWORK 10
gvl_ribmachine.ReadyToCut := gvl_ribmachine.InCycle AND clampclosed OR gvl_ribmachine.ReadyToCut AND NOT GVL_RibMachine.CutComplete;

// NETWORK 11
_w1 := gvl_ribmachine.InCycle AND clampclosed AND GVL_RibMachine.MeasureComplete AND NOT GVL_RibMachine.RibMachineFaulted OR GVL_RibMachine.SawStart AND NOT GVL_RibMachine.CutComplete OR gvl_hmi.ManualMode AND gvl_saf.SafetyOk AND Outputs_RB.HmiPBSawStart AND NOT Outputs_RB.HmiPBSawStop;
DustCollectStartRequest := _w1;
StartSawRequest := _w1;

// NETWORK 12: Wait to traverse to ensure motor is up to speed before cutting.
SawDwellTimer(IN := GVL_RibMachine.SawStart, PT := T#750ms, ET => SawDwellTimerElapsed); // TON
SawDwellDoneBit := SawDwellTimer.Q;

// NETWORK 13
// Wait a half second to make sure motor is running
TraverseDwellTimer(
    IN := GVL_RibMachine.TraverseStartFwd OR GVL_RibMachine.TraverseStartRev,
    PT := T#500ms,
    ET => TraverseDwellTimerElapsed); // TON
TraverseDwellDoneBit := TraverseDwellTimer.Q;

// NETWORK 14
GVL_RibMachine.TraverseStartFwd := (gvl_ribmachine.InCycle AND clampclosed AND GVL_RibMachine.MeasureComplete AND GVL_RibMachine.SawStart AND SawDwellDoneBit OR GVL_RibMachine.TraverseStartFwd AND NOT GVL_RibMachine.CutComplete AND NOT GVL_RibMachine.TraverseStartRev OR gvl_hmi.ManualMode AND gvl_saf.SafetyOk AND Outputs_RB.HmiPBTraverseFwd AND NOT Outputs_RB.HmiPBTraverseRev) AND NOT GVL_RibMachine.SawExtendedOn AND NOT GVL_RibMachine.RibMachineFaulted;

// NETWORK 15
_rt3(CLK := GVL_RibMachine.SawExtendedOn);
GVL_RibMachine.TraverseStartRev := (gvl_ribmachine.InCycle AND clampclosed AND SawTraversing AND _rt3.Q OR GVL_RibMachine.TraverseStartRev AND NOT SawHome OR gvl_hmi.ManualMode AND gvl_saf.SafetyOk AND Outputs_RB.HmiPBTraverseRev AND NOT Outputs_RB.HmiPBTraverseFwd) AND NOT GVL_RibMachine.RibMachineFaulted;

END_PROGRAM

// ---- Machine System/PRGs/Rib Machine/Outputs_RB.TcPOU
PROGRAM Outputs_RB
VAR
	HmiPBDoorRequest: BOOL;
	HmiPBIndexFwd: BOOL;
	HmiPBIndexRev: BOOL;
	HmiPBDustCollect: BOOL;
	HmiPBSawStart: BOOL;
	HmiPBSawStop: BOOL;
	HmiPBTraverseFwd: BOOL;
	HmiPBTraverseRev: BOOL;
	HmiPBLiftRaise: BOOL;
	HmiPBLiftLower: BOOL;
	HmiPBTransferFwd: BOOL;
	HmiPBTransferRev: BOOL;
	HmiPBTransferClampOpen: BOOL;
	HmiPBTransferClampClose: BOOL;
	HmiPBTransferClampFwd: BOOL;
	HmiPBTransferClampRev: BOOL;
	HmiPBSawClampClose: BOOL;
	HmiPBSawClampOpen: BOOL;
	HmiPBSawClampFwd: BOOL;
	HmiPBSawClampRev: BOOL;
	HmiPBPinsRaise: BOOL;
	HmiPBPinsLower: BOOL;
	
	
	
	
END_VAR

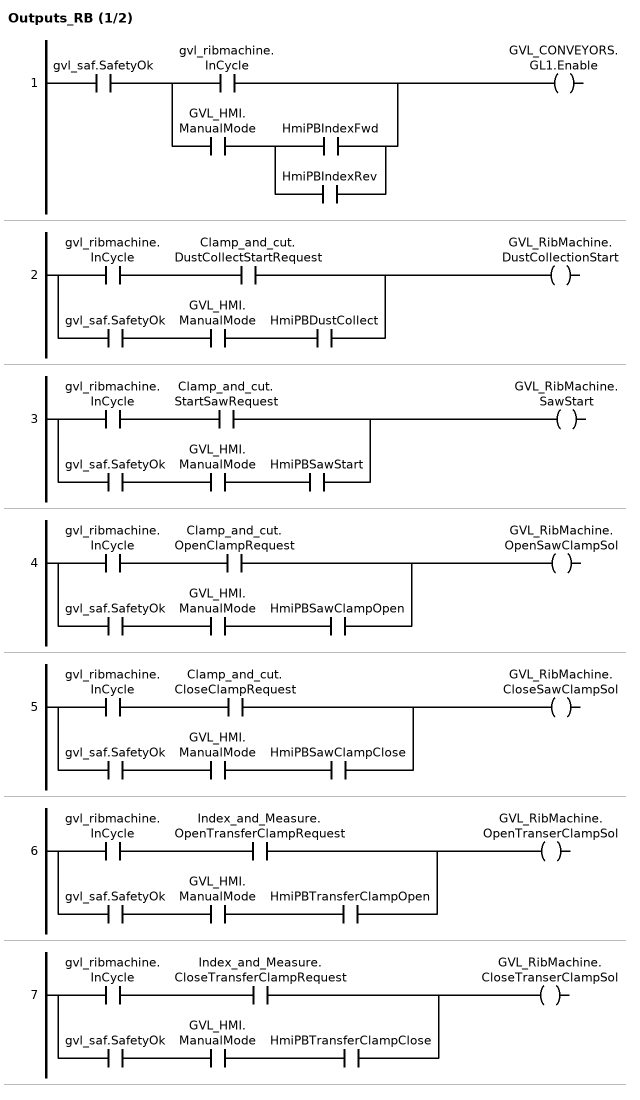
// NETWORK 1
GVL_CONVEYORS.GL1.Enable := gvl_saf.SafetyOk AND (gvl_ribmachine.InCycle OR GVL_HMI.ManualMode AND (HmiPBIndexFwd OR HmiPBIndexRev));

// NETWORK 2
GVL_RibMachine.DustCollectionStart := gvl_ribmachine.InCycle AND Clamp_and_cut.DustCollectStartRequest OR gvl_saf.SafetyOk AND GVL_HMI.ManualMode AND HmiPBDustCollect;

// NETWORK 3
GVL_RibMachine.SawStart := gvl_ribmachine.InCycle AND Clamp_and_cut.StartSawRequest OR gvl_saf.SafetyOk AND GVL_HMI.ManualMode AND HmiPBSawStart;

// NETWORK 4
GVL_RibMachine.OpenSawClampSol := gvl_ribmachine.InCycle AND Clamp_and_cut.OpenClampRequest OR gvl_saf.SafetyOk AND GVL_HMI.ManualMode AND HmiPBSawClampOpen;

// NETWORK 5
GVL_RibMachine.CloseSawClampSol := gvl_ribmachine.InCycle AND Clamp_and_cut.CloseClampRequest OR gvl_saf.SafetyOk AND GVL_HMI.ManualMode AND HmiPBSawClampClose;

// NETWORK 6
GVL_RibMachine.OpenTranserClampSol := gvl_ribmachine.InCycle AND Index_and_Measure.OpenTransferClampRequest OR gvl_saf.SafetyOk AND GVL_HMI.ManualMode AND HmiPBTransferClampOpen;

// NETWORK 7
GVL_RibMachine.CloseTranserClampSol := gvl_ribmachine.InCycle AND Index_and_Measure.CloseTransferClampRequest OR gvl_saf.SafetyOk AND GVL_HMI.ManualMode AND HmiPBTransferClampClose;

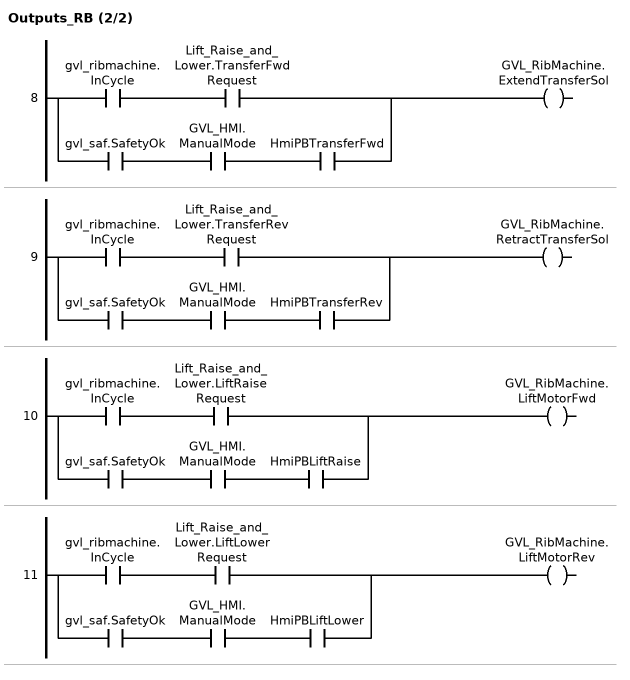
// NETWORK 8
GVL_RibMachine.ExtendTransferSol := gvl_ribmachine.InCycle AND Lift_Raise_and_Lower.TransferFwdRequest OR gvl_saf.SafetyOk AND GVL_HMI.ManualMode AND HmiPBTransferFwd;

// NETWORK 9
GVL_RibMachine.RetractTransferSol := gvl_ribmachine.InCycle AND Lift_Raise_and_Lower.TransferRevRequest OR gvl_saf.SafetyOk AND GVL_HMI.ManualMode AND HmiPBTransferRev;

// NETWORK 10
GVL_RibMachine.LiftMotorFwd := gvl_ribmachine.InCycle AND Lift_Raise_and_Lower.LiftRaiseRequest OR gvl_saf.SafetyOk AND GVL_HMI.ManualMode AND HmiPBLiftRaise;

// NETWORK 11
GVL_RibMachine.LiftMotorRev := gvl_ribmachine.InCycle AND Lift_Raise_and_Lower.LiftLowerRequest OR gvl_saf.SafetyOk AND GVL_HMI.ManualMode AND HmiPBLiftLower;

END_PROGRAM

// ---- Machine System/PRGs/Rib Machine/Lift_Raise_and_Lower.TcPOU
PROGRAM Lift_Raise_and_Lower
VAR
	LiftRaiseRequest: BOOL; // Logic bit to request transfer move forward towards lift bed.
	LiftLowerRequest: BOOL; // Logic bit to request transfer move reverse towards home switch
	ReadyToRaise:BOOL; // Logic bit to indicate ready to lift
	ReadyToLower:BOOL; // Logic bit to indicate ready to lower
	OpenTransferClampRequest:BOOL; // Logic bit to request transfer clamp open
	CloseTransferClampRequest:BOOL; // Logic bit to request transfer clamp close
	TransferFwdRequest: BOOL; // Logic bit to request transfer move forward towards lift bed.
	TransferRevRequest: BOOL; // Logic bit to request transfer move reverse towards home switch
	RibsReadyForPickup:BOOL; // Hoist is up and ribs have been cut to lenght, waiting for gripper to acknowledge pick up
	
END_VAR

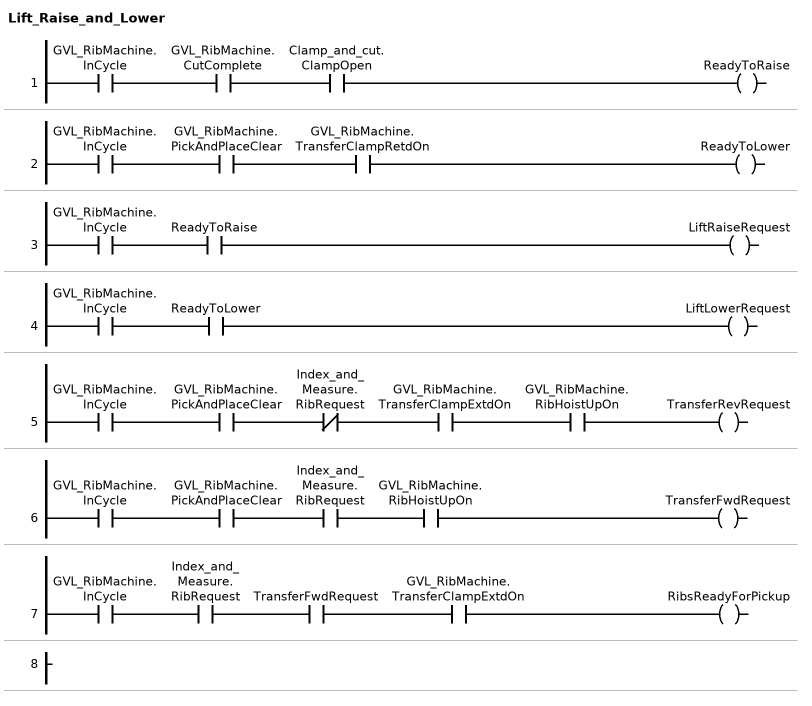
// NETWORK 1
ReadyToRaise := GVL_RibMachine.InCycle AND GVL_RibMachine.CutComplete AND Clamp_and_cut.ClampOpen;

// NETWORK 2
ReadyToLower := GVL_RibMachine.InCycle AND GVL_RibMachine.PickAndPlaceClear AND GVL_RibMachine.TransferClampRetdOn;

// NETWORK 3
LiftRaiseRequest := GVL_RibMachine.InCycle AND ReadyToRaise;

// NETWORK 4
LiftLowerRequest := GVL_RibMachine.InCycle AND ReadyToLower;

// NETWORK 5
TransferRevRequest := GVL_RibMachine.InCycle AND GVL_RibMachine.PickAndPlaceClear AND NOT Index_and_Measure.RibRequest AND GVL_RibMachine.TransferClampExtdOn AND GVL_RibMachine.RibHoistUpOn;

// NETWORK 6
TransferFwdRequest := GVL_RibMachine.InCycle AND GVL_RibMachine.PickAndPlaceClear AND Index_and_Measure.RibRequest AND GVL_RibMachine.RibHoistUpOn;

// NETWORK 7
RibsReadyForPickup := GVL_RibMachine.InCycle AND Index_and_Measure.RibRequest AND TransferFwdRequest AND GVL_RibMachine.TransferClampExtdOn;

// NETWORK 8

END_PROGRAM

// ---- Machine System/PRGs/Rib Machine/Fault_Logic.TcPOU
PROGRAM Fault_Logic
VAR
	
	ScrapBinFullWarning: BOOL;
	RibHopperEmptyFault: BOOL;
	RibHopperNearEmptyWarning: BOOL;
	RibMeasureFault: BOOL;
	LowAirPresFault: BOOL;
	GuardOpenFault: BOOL;
	MotorFault: BOOL;
	JamFault: BOOL;
	AirPresTon : TON;
	AirPresElapsed: TIME;
	
	
	
END_VAR

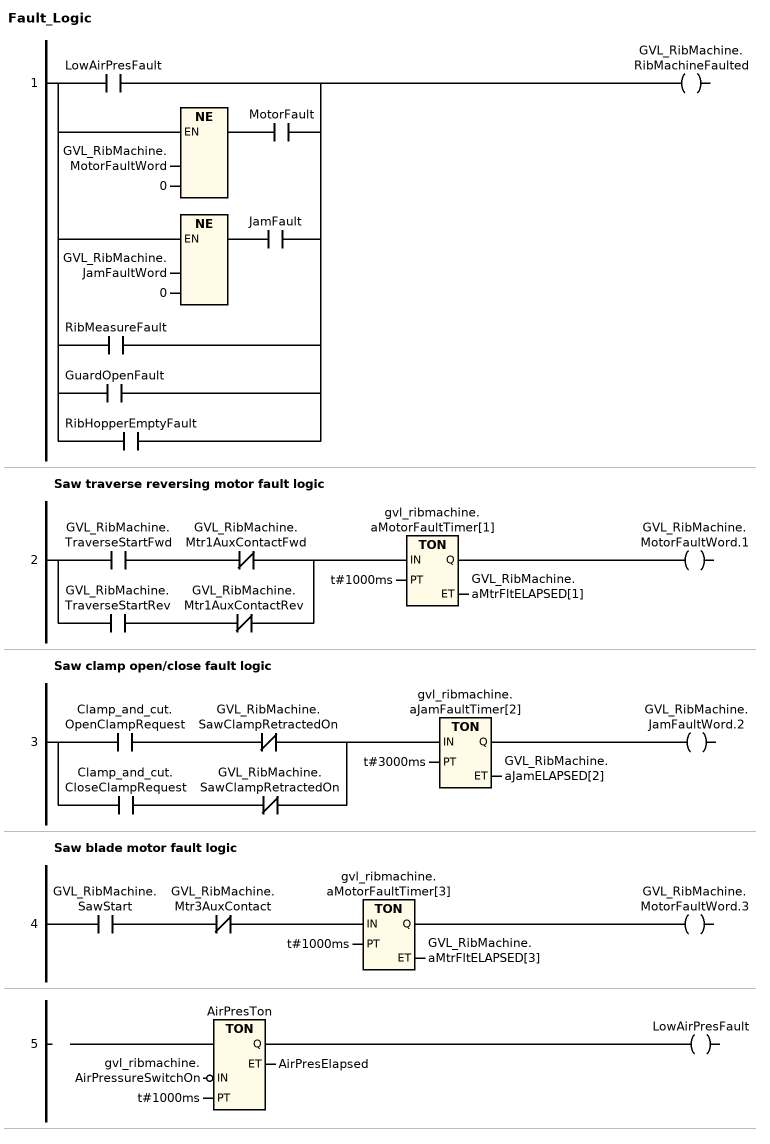
// NETWORK 1
GVL_RibMachine.RibMachineFaulted := LowAirPresFault OR GVL_RibMachine.MotorFaultWord <> 0 AND MotorFault OR GVL_RibMachine.JamFaultWord <> 0 AND JamFault OR RibMeasureFault OR GuardOpenFault OR RibHopperEmptyFault;

// NETWORK 2: Saw traverse reversing motor fault logic
gvl_ribmachine.aMotorFaultTimer[1](
    IN := GVL_RibMachine.TraverseStartFwd AND NOT GVL_RibMachine.Mtr1AuxContactFwd OR GVL_RibMachine.TraverseStartRev AND NOT GVL_RibMachine.Mtr1AuxContactRev,
    PT := t#1000ms,
    ET => GVL_RibMachine.aMtrFltELAPSED[1]); // TON
GVL_RibMachine.MotorFaultWord.1 := gvl_ribmachine.aMotorFaultTimer[1].Q;

// NETWORK 3: Saw clamp open/close fault logic
gvl_ribmachine.aJamFaultTimer[2](
    IN := Clamp_and_cut.OpenClampRequest AND NOT GVL_RibMachine.SawClampRetractedOn OR Clamp_and_cut.CloseClampRequest AND NOT GVL_RibMachine.SawClampRetractedOn,
    PT := t#3000ms,
    ET => GVL_RibMachine.aJamELAPSED[2]); // TON
GVL_RibMachine.JamFaultWord.2 := gvl_ribmachine.aJamFaultTimer[2].Q;

// NETWORK 4: Saw blade motor fault logic
gvl_ribmachine.aMotorFaultTimer[3](
    IN := GVL_RibMachine.SawStart AND NOT GVL_RibMachine.Mtr3AuxContact,
    PT := t#1000ms,
    ET => GVL_RibMachine.aMtrFltELAPSED[3]); // TON
GVL_RibMachine.MotorFaultWord.3 := gvl_ribmachine.aMotorFaultTimer[3].Q;

// NETWORK 5
AirPresTon(IN := NOT gvl_ribmachine.AirPressureSwitchOn, PT := t#1000ms, ET => AirPresElapsed); // TON
LowAirPresFault := AirPresTon.Q;

END_PROGRAM

// ---- Machine System/PRGs/Rib Machine/Interlocks_to_Main_Line.TcPOU
PROGRAM Interlocks_to_Main_Line
VAR
	RibMachineReady: BOOL;
	
	
	
END_VAR

// NETWORK 1

END_PROGRAM

// ---- Machine System/PRGs/ALARM AND STATUS/SYSTEM.TcPOU
PROGRAM SYSTEM
VAR
	fbGetCurTaskIdx  : GETCURTASKINDEX; // PlcTaskSystemInfo for Cycle time
	
	
END_VAR

fbGetCurTaskIdx();
GVL.CycleTime := _TaskInfo[fbGetCurTaskIdx.index].CycleTime/10000;

GVL.GetLocalSystemTimeFB(
	sNetID:= , 
	bEnable:= TRUE, 
	dwCycle:= 1, 
	dwOpt:= , 
	tTimeout:= , 
	bValid=> , 
	systemTime=> , 
	tzID=> );
	
GVL.SystemDateTime := SYSTEMTIME_TO_STRING(GVL.GetLocalSystemTimeFB.systemTime);

GVL.SystemDate := MID(STR:=GVL.SystemDateTime , LEN:=10 , POS:=1 );
GVL.SystemTime := MID(STR:=GVL.SystemDateTime , LEN:=8 , POS:=12 );

END_PROGRAM

// ---- CNC HMI/P_GFunctionMonitor_2.TcPOU
PROGRAM P_GFunctionMonitor_2
VAR
	bReadGcode: BOOL;
	fbADSRead: ADSREADEX;
	GBuffer: ARRAY[1..39]OF WORD;
	nPathPrep: WORD;
	nPlane: WORD;
	nCutterComp: WORD;
	nDeselectDiamProg: WORD;
	nZeroOffset: WORD;
	nContMode: WORD;
	nMeasureMode: WORD;
	nDeselectSpline: WORD;
	nDeselectCornerRed: WORD;
	//toString
		sPathPrep: STRING;
		sPlane: STRING;
		sCutterComp: STRING;
		sDeselectDiamProg: STRING;
		sZeroOffset: STRING;
		sContMode: STRING;
		sMeasureMode: STRING;
		sDeselectSpline: STRING;
		sDeselectCornerRed: STRING;
	fbUpdate: TON;
	sLocalAmsNet 	: STRING; 
	getAmsNet : FB_GetLocalAmsNetId;
	bLocalAmsNet : BOOL;
	
	sGCodeOut : string;
END_VAR

//Read active G code
IF sLocalAmsNet ='' THEN
	bLocalAmsNet := TRUE;
ELSE
	blocalamsNet := FALSE;
END_IF
getAmsNet(bExecute:=bLocalAmsNet, tTimeOut:=DEFAULT_ADS_TIMEOUT,AddrString => sLocalAmsNet);

IF Global_HMI.PLCSelectedChannel = 1 THEN //set this to the selected channel and duplicate for as many channels as necessary
	bReadGcode := TRUE;
	ELSE breadgcode := FALSE;
END_IF

fbUpdate.PT := T#1S;
IF bReadGcode THEN
	fbUpdate.IN := TRUE;
ELSE
	fbUpdate.IN := FALSE;
END_IF

IF fbUpdate.Q THEN
	fbADSRead(
	NETID:=sLocalAmsNet, 
	PORT:=553, 
	IDXGRP:=16#120102, //120102 for ch2 active g code {120101 for ch1}
	IDXOFFS:=16#3C, 
	LEN:=SIZEOF(GBuffer), 
	DESTADDR:=ADR(GBuffer), 
	READ:=TRUE, 
	TMOUT:=T#2S, 
	BUSY=> , 
	ERR=> , 
	ERRID=> , 
	COUNT_R=> );
	
	IF NOT fbADSRead.BUSY THEN
		fbADSRead(
			NETID:=sLocalAmsNet, 
			PORT:=553, 
			IDXGRP:=16#120101, 
			IDXOFFS:=16#3C, 
			LEN:=SIZEOF(GBuffer), 
			DESTADDR:=ADR(GBuffer), 
			READ:=FALSE, 
			TMOUT:=T#2S);
		fbUpdate.IN := FALSE;
	END_IF
END_IF
//Parse them out
nPathPrep 			:= GBuffer[1];
nPlane 				:= GBuffer[5];
nCutterComp 		:= GBuffer[8];
nDeselectDiamProg 	:= GBuffer[9];
nZeroOffset 		:= GBuffer[10];
nContMode			:= GBuffer[11];
nMeasureMode 		:= GBuffer[15];
nDeselectSpline 	:= GBuffer[30];
nDeselectCornerRed 	:= GBuffer[32];
//to string
IF 	nPathPrep > 0 AND npathprep< 65535 THEN
	sPathPrep:= concat(concat('G',TO_STRING(nPathPrep)),' '); ELSE sPathPrep :=''; END_IF
IF nPlane >0 AND nPlane<65535 THEN
	sPlane:= concat(concat('G',TO_STRING(nPlane)),' '); ELSE sPlane:=''; END_IF
IF nCutterComp>0 AND nCutterComp<65535 THEN
	sCutterComp:= concat(concat('G',TO_STRING(nCutterComp)),' '); ELSE sCutterComp :=''; END_IF
IF nDeselectDiamProg >0 AND nDeselectDiamProg<65535 THEN
	sDeselectDiamProg:= concat(concat('G',TO_STRING(nDeselectDiamProg)),' '); ELSE sDeselectDiamProg :=''; END_IF
IF nZeroOffset >0 AND nZeroOffset<65535 THEN
	sZeroOffset:= concat(concat('G',TO_STRING(nZeroOffset)),' '); ELSE sZeroOffset:=''; END_IF
IF ncontmode > 0 AND ncontmode < 65535 THEN
	sContMode:= concat(concat('G',TO_STRING(nContMode)),' '); ELSE scontmode:=''; END_IF
IF nMeasureMode >0 AND nMeasureMode < 65535 THEN
	sMeasureMode:= concat(concat('G',TO_STRING(nMeasureMode)),' '); ELSE sMeasureMode := ''; END_IF
IF 	nDeselectSpline > 0 AND nDeselectSpline< 65535 THEN
	sDeselectSpline:= concat(concat('G',TO_STRING(nDeselectSpline)),' '); ELSE sDeselectSpline:=''; END_IF
IF nDeselectCornerRed >0 AND nDeselectCornerRed < 65535 THEN
	sDeselectCornerRed:= concat(concat('G',TO_STRING(nDeselectCornerRed)),' '); ELSE sDeselectCornerRed:=''; END_IF
//sGCodeOut := Concat(Concat(CONCAT('G',nPathPrep),' G'),nPlane);
sGCodeOut := Concat(Concat(Concat(Concat(Concat(Concat(Concat(Concat(sPathPrep,sPlane),sCutterComp),sDeselectDiamProg),sZeroOffset),sContMode),sMeasureMode),sDeselectSpline),sDeselectCornerRed);

//Timer
fbUpdate();

END_PROGRAM

// ---- Machine System/FUNCTIONS/F_CheckRollerDoor.TcPOU
FUNCTION F_CheckRollerDoor : BOOL
VAR_INPUT
	CurrentPos 		: REAL;
	RequestedPos 	: REAL;
	Door 			: sRollerDoor;
END_VAR
VAR
	DoorPos : REAL := 100000;
END_VAR

IF (CurrentPos < DoorPos AND RequestedPos > DoorPos) OR (CurrentPos > DoorPos AND RequestedPos < DoorPos) THEN
	Door.AutoOpenRequest := 1;
	IF Door.StatusOpenedInput THEN
		F_CheckRollerDoor := 1;
	END_IF
	ELSE
	F_CheckRollerDoor := 1;	
END_IF

END_FUNCTION

// ---- Machine System/FUNCTIONS/F_PartIsClamped.TcPOU
FUNCTION F_PartIsClamped : BOOL
VAR_INPUT
	WX : sBogie;
END_VAR
VAR
END_VAR

IF (WX.A.bClamped AND WX.B.bClamped) OR NOT(WX.bEnabled) THEN
	F_PartIsClamped := 1;
	ELSE
		F_PartIsClamped := 0;
END_IF

END_FUNCTION

// ---- Machine System/PRGs/ALARM AND STATUS/Database_PRG_SEQUENCE_1.TcPOU
PROGRAM Database_PRG_SEQUENCE_1
VAR
	Process			: ARRAY [1..MAX_DBCOLUMNS] OF ST_Process;
	fbSQLDatabase	: FB_SQLDatabaseEvt(sNetID :='192.168.0.136.1.1', tTimeout := T#5S);
	fbSQLCommand	: FB_SQLCommandEvt(sNetID :='192.168.0.136.1.1', tTimeout := T#5S);
	step			: INT := 10;
	CMD_1			: STRING(5000);
	CMD_2			: STRING(5000);
	CMD_3			: STRING(5000);
	CMD_4			: STRING(5000);
	sCMD			: STRING(5000);
	sCMD1			: STRING(5000);
	sCMD2			: STRING(5000);
	EventID			: INT;
	EventString		: STRING(5000);
	
			
END_VAR

CASE step OF
	
10: //OPEN CONNECTION
	IF fbSQLDatabase.Connect(1) THEN
		step := step + 10;
	END_IF

20: //CREATE COMMAND 
	IF fbSQLDatabase.CreateCmd(ADR(fbSQLCommand)) THEN
		step := step + 10;
	END_IF

30: //INSERT COMMAND
	CMD_1	:= 'INSERT INTO MixerTable (EventTime, EventID, EventString) VALUES (';
	CMD_2	:= 'DATETIME(),';
	CMD_3	:= ')';
	sCMD	:= CONCAT (CMD_1, CONCAT(CMD_2,CONCAT (CONCAT ('$'',INT_TO_STRING(EventID)),'$',')));
	sCMD1	:= CONCAT (sCMD, CONCAT(CONCAT('$'', EventString), '$''));
	sCMD2	:= CONCAT (sCMD1, CMD_3);
	IF fbSQLCommand.Execute(ADR(sCMD2), SIZEOF(sCMD2)) THEN
		step := step + 1000;
	END_IF
	
1030: //CLOSE CONNECTION
	IF fbSQLDatabase.Disconnect() THEN
		step := step + 1;
	END_IF
		
END_CASE

END_PROGRAM

// ---- Machine System/PRGs/ALARM AND STATUS/Light.TcPOU
PROGRAM Light
VAR
	Bulk1LightFB : LightFB;
	Bulk2LightFB : LightFB;
	BulkResinLightFB : LightFB;
	Filter1LightFB : LightFB;
	Filter2LightFB : LightFB;
	Filter3LightFB : LightFB;
	Filter4LightFB : LightFB;
	
	//Lights
	Bulk1Light : StackLight;
	Bulk2Light : StackLight;
	BulkResinLight : StackLight;
	Filter1Light : StackLight;
	Filter2Light : StackLight;
	Filter3Light : StackLight;
	Filter4Light : StackLight;
	

END_VAR

Bulk1LightFB(
	Red := Bulk1Light.Red,
	Yellow := Bulk1Light.Yellow,
	Green := Bulk1Light.Green,
	BuzzerOnInput := Bulk1Light.BuzzerOnInput,
	BuzzerStyleInput := Bulk1Light.BuzzerStyleInput
	);
	
	Bulk1Light.LED_A := Bulk1LightFB.LED_A;
	Bulk1Light.LED_B := Bulk1LightFB.LED_B;
	Bulk1Light.LED_C := Bulk1LightFB.LED_C;
	Bulk1Light.BuzzerOnOutput := Bulk1LightFB.BuzzerOnOutput;
	Bulk1Light.BuzzerStyleOutput := Bulk1LightFB.BuzzerStyleOutput;
	
Bulk2LightFB(
	Red := Bulk2Light.Red,
	Yellow := Bulk2Light.Yellow,
	Green := Bulk2Light.Green,
	BuzzerOnInput := Bulk2Light.BuzzerOnInput,
	BuzzerStyleInput := Bulk2Light.BuzzerStyleInput
	);
	
	Bulk2Light.LED_A := Bulk2LightFB.LED_A;
	Bulk2Light.LED_B := Bulk2LightFB.LED_B;
	Bulk2Light.LED_C := Bulk2LightFB.LED_C;
	Bulk2Light.BuzzerOnOutput := Bulk2LightFB.BuzzerOnOutput;
	Bulk2Light.BuzzerStyleOutput := Bulk2LightFB.BuzzerStyleOutput;

BulkResinLightFB(
	Red := BulkResinLight.Red,
	Yellow := BulkResinLight.Yellow,
	Green := BulkResinLight.Green,
	BuzzerOnInput := BulkResinLight.BuzzerOnInput,
	BuzzerStyleInput := BulkResinLight.BuzzerStyleInput
	);
	
	BulkResinLight.LED_A := BulkResinLightFB.LED_A;
	BulkResinLight.LED_B := BulkResinLightFB.LED_B;
	BulkResinLight.LED_C := BulkResinLightFB.LED_C;
	BulkResinLight.BuzzerOnOutput := BulkResinLightFB.BuzzerOnOutput;
	BulkResinLight.BuzzerStyleOutput := BulkResinLightFB.BuzzerStyleOutput;

Filter1LightFB(
	Red := Filter1Light.Red,
	Yellow := Filter1Light.Yellow,
	Green := Filter1Light.Green,
	BuzzerOnInput := Filter1Light.BuzzerOnInput,
	BuzzerStyleInput := Filter1Light.BuzzerStyleInput
	);
	
	Filter1Light.LED_A := Filter1LightFB.LED_A;
	Filter1Light.LED_B := Filter1LightFB.LED_B;
	Filter1Light.LED_C := Filter1LightFB.LED_C;
	Filter1Light.BuzzerOnOutput := Filter1LightFB.BuzzerOnOutput;
	Filter1Light.BuzzerStyleOutput := Filter1LightFB.BuzzerStyleOutput;

Filter2LightFB(
	Red := Filter2Light.Red,
	Yellow := Filter2Light.Yellow,
	Green := Filter2Light.Green,
	BuzzerOnInput := Filter2Light.BuzzerOnInput,
	BuzzerStyleInput := Filter2Light.BuzzerStyleInput
	);
	
	Filter2Light.LED_A := Filter2LightFB.LED_A;
	Filter2Light.LED_B := Filter2LightFB.LED_B;
	Filter2Light.LED_C := Filter2LightFB.LED_C;
	Filter2Light.BuzzerOnOutput := Filter2LightFB.BuzzerOnOutput;
	Filter2Light.BuzzerStyleOutput := Filter2LightFB.BuzzerStyleOutput;

Filter3LightFB(
	Red := Filter3Light.Red,
	Yellow := Filter3Light.Yellow,
	Green := Filter3Light.Green,
	BuzzerOnInput := Filter3Light.BuzzerOnInput,
	BuzzerStyleInput := Filter3Light.BuzzerStyleInput
	);
	
	Filter3Light.LED_A := Filter3LightFB.LED_A;
	Filter3Light.LED_B := Filter3LightFB.LED_B;
	Filter3Light.LED_C := Filter3LightFB.LED_C;
	Filter3Light.BuzzerOnOutput := Filter3LightFB.BuzzerOnOutput;
	Filter3Light.BuzzerStyleOutput := Filter3LightFB.BuzzerStyleOutput;

Filter4LightFB(
	Red := Filter4Light.Red,
	Yellow := Filter4Light.Yellow,
	Green := Filter4Light.Green,
	BuzzerOnInput := Filter4Light.BuzzerOnInput,
	BuzzerStyleInput := Filter4Light.BuzzerStyleInput
	);
	
	Filter4Light.LED_A := Filter4LightFB.LED_A;
	Filter4Light.LED_B := Filter4LightFB.LED_B;
	Filter4Light.LED_C := Filter4LightFB.LED_C;
	Filter4Light.BuzzerOnOutput := Filter4LightFB.BuzzerOnOutput;
	Filter4Light.BuzzerStyleOutput := Filter4LightFB.BuzzerStyleOutput;
	
	
	
	
IF NewBatch.ResinTote.ActualScaleWeight < 400 AND NewBatch.ResinTote.ActualScaleWeight > 50 THEN
	BulkResinLight.Green := 0;
	BulkResinLight.Yellow := 1;
END_IF

IF NewBatch.ResinTote.ActualScaleWeight < 210 THEN
	BulkResinLight.Yellow := 0;
	BulkResinLight.Red := 1;
END_IF

IF NewBatch.ResinTote.ActualScaleWeight > 400 THEN
	BulkResinLight.Yellow := 0;
	BulkResinLight.Red := 0;
	BulkResinLight.Green := 1;
END_IF

//Filter 1 Light Control
	IF HMI.Filter1Runtime >= HMI.FilterRuntimeAlarmTimeInput THEN
		//Raise Filter 1 Alarm
		Filter1Light.Red := 1; //Turn Red Light on 
		Filter1Light.BuzzerOnInput := 1; // Turn Buzzer On
		Filter1Light.Yellow := 0;
	ELSIF TIME_TO_DINT(HMI.Filter1Runtime) > TIME_TO_DINT(HMI.FilterRuntimeAlarmTimeInput)*3/4 AND TIME_TO_DINT(HMI.Filter1Runtime) < TIME_TO_DINT(HMI.FilterRuntimeAlarmTimeInput) THEN
		Filter1Light.Yellow := 1; //Turn Yellow Light on at 75% filter usage
	ELSE
		Filter1Light.Red := 0; 
		Filter1Light.BuzzerOnInput := 0; 
		Filter1Light.Yellow := 0; 
	END_IF
	
//Filter 2 Light Control
	IF HMI.Filter2Runtime >= HMI.FilterRuntimeAlarmTimeInput THEN
		//Raise Filter 2 Alarm
		Filter2Light.Red := 1; //Turn Red Light on 
		Filter2Light.BuzzerOnInput := 1; // Turn Buzzer On
		Filter2Light.Yellow := 0;
	ELSIF TIME_TO_DINT(HMI.Filter2Runtime) > TIME_TO_DINT(HMI.FilterRuntimeAlarmTimeInput)*3/4 AND TIME_TO_DINT(HMI.Filter2Runtime) < TIME_TO_DINT(HMI.FilterRuntimeAlarmTimeInput) THEN
		Filter2Light.Yellow := 1; //Turn Yellow Light on at 75% filter usage
	ELSE
		Filter2Light.Red := 0; 
		Filter2Light.BuzzerOnInput := 0; 
		Filter2Light.Yellow := 0; 
	END_IF	
	
//Filter 3 Light Control
	IF HMI.Filter3Runtime >= HMI.FilterRuntimeAlarmTimeInput THEN
		//Raise Filter 3 Alarm
		Filter3Light.Red := 1; //Turn Red Light on 
		Filter3Light.BuzzerOnInput := 1; // Turn Buzzer On
		Filter3Light.Yellow := 0;
	ELSIF TIME_TO_DINT(HMI.Filter3Runtime) > TIME_TO_DINT(HMI.FilterRuntimeAlarmTimeInput)*3/4 AND TIME_TO_DINT(HMI.Filter3Runtime) < TIME_TO_DINT(HMI.FilterRuntimeAlarmTimeInput) THEN
		Filter3Light.Yellow := 1; //Turn Yellow Light on at 75% filter usage
	ELSE
		Filter3Light.Red := 0; 
		Filter3Light.BuzzerOnInput := 0; 
		Filter3Light.Yellow := 0; 
	END_IF	
//Filter 4 Light Control
	IF HMI.Filter4Runtime >= HMI.FilterRuntimeAlarmTimeInput THEN
		//Raise Filter 4 Alarm
		Filter4Light.Red := 1; //Turn Red Light on 
		Filter4Light.BuzzerOnInput := 1; // Turn Buzzer On
		Filter4Light.Yellow := 0;
	ELSIF TIME_TO_DINT(HMI.Filter4Runtime) > TIME_TO_DINT(HMI.FilterRuntimeAlarmTimeInput)*3/4 AND TIME_TO_DINT(HMI.Filter4Runtime) < TIME_TO_DINT(HMI.FilterRuntimeAlarmTimeInput) THEN
		Filter4Light.Yellow := 1; //Turn Yellow Light on at 75% filter usage
	ELSE
		Filter4Light.Red := 0; 
		Filter4Light.BuzzerOnInput := 0; 
		Filter4Light.Yellow := 0; 
	END_IF

END_PROGRAM

// ---- Machine System/PRGs/ALARM AND STATUS/PumpStatus.TcPOU
PROGRAM PumpStatus
VAR
	
	Pump1RuntimeFB : RunTimetracker;
	Pump2RuntimeFB : RunTimetracker;
	Pump3RuntimeFB : RunTimetracker;
	Pump4RuntimeFB : RunTimetracker;
	
END_VAR

// Link Pump status with HMI GVL

	HMI.Pump1.PumpOn	:=	Resin.Pump1.PumpOn;
	HMI.Pump2.PumpOn	:=	Resin.Pump2.PumpOn;
	HMI.Pump3.PumpOn	:=	Resin.Pump3.PumpOn;
	HMI.Pump4.PumpOn	:=	Resin.Pump4.PumpOn;
		
// Runtime Tracking Function block calls for Pumps
	Pump1RuntimeFB(RunTimerStartSignal:=IO.Pump1On , Reset:=HMI.Pump1.RuntimeResetButton, RunTime=>HMI.Pump1Runtime);
	Pump2RuntimeFB(RunTimerStartSignal:=IO.Pump2On , Reset:=HMI.Pump2.RuntimeResetButton, RunTime=>HMI.Pump2Runtime);
	Pump3RuntimeFB(RunTimerStartSignal:=IO.Pump3On , Reset:=HMI.Pump3.RuntimeResetButton, RunTime=>HMI.Pump3Runtime);
	Pump4RuntimeFB(RunTimerStartSignal:=IO.Pump4On , Reset:=HMI.Pump4.RuntimeResetButton, RunTime=>HMI.Pump4Runtime);
// Runtime Alarms for Pump Usage
	//Pump 1
	IF HMI.Pump1Runtime >= HMI.Pump1.RuntimeAlarmTimeInput THEN
		HMI.Pump1.ChangeOutNeededAlarm := 1;
		//Eventlog Message pump 1 needs changout
	ELSE
		HMI.Pump1.ChangeOutNeededAlarm := 0;
	END_IF
	//Pump 2
	IF HMI.Pump2Runtime >= HMI.Pump2.RuntimeAlarmTimeInput THEN
		HMI.Pump2.ChangeOutNeededAlarm := 1;
		//Eventlog Message pump 2 needs changout
	ELSE
		HMI.Pump2.ChangeOutNeededAlarm := 0;
	END_IF
	//Pump 3
	IF HMI.Pump3Runtime >= HMI.Pump3.RuntimeAlarmTimeInput THEN
		HMI.Pump3.ChangeOutNeededAlarm := 1;
		//Eventlog Message pump 3 needs changout
	ELSE
		HMI.Pump3.ChangeOutNeededAlarm := 0;
	END_IF
	//Pump 4
	IF HMI.Pump4Runtime >= HMI.Pump4.RuntimeAlarmTimeInput THEN
		HMI.Pump4.ChangeOutNeededAlarm := 1;
		//Eventlog Message pump 4 needs changout
	ELSE
		HMI.Pump4.ChangeOutNeededAlarm := 0;
	END_IF
	
	// Manual Req Block Control - Turn Visiblity off when not in individual valve control
	IF resin.ManualFlowState <> 70 THEN
		HMI.Pump1.ManualRequestOn := HMI.Pump1.PumpOn;
		HMI.Pump2.ManualRequestOn := HMI.Pump2.PumpOn;
		HMI.Pump3.ManualRequestOn := HMI.Pump3.PumpOn;
		HMI.Pump4.ManualRequestOn := HMI.Pump4.PumpOn;
	END_IF

END_PROGRAM

// ---- Machine System/PRGs/CAM_CNC/Gun/myCounter.TcPOU
PROGRAM myCounter
VAR
	
	iPumpCount AT %I* : UDINT;
	iGunRPMCount AT %I* : UDINT;
	iLastGunRPMCount : UDINT;
	
END_VAR

//plug both into EL1512 
//count chopper gun rpm (rising trigger)
	//add rpm hmi display (floating average)
IF iGunRPMCount <> iLastGunRPMCount THEN
	iLastGunRPMCount := iGunRPMCount;
END_IF
//count resin/mek pump strokes (rising trigger)
	//add flow rate hmi display (floating average)

END_PROGRAM

// ---- Machine System/PRGs/CAM_CNC/Gun/myGun.TcPOU
PROGRAM myGun
VAR
	iFiberPres AT %Q* : UINT;
	bFiberOn : BOOL;
	bManualChop : BOOL;
	iFiberScale : UINT;
END_VAR

iFiberScale := PLCSpindleOverride;

IF GVL_IO.bSprayOn = TRUE AND bFiberOn THEN
	iFiberPres :=32000 *iFiberScale/100;
	ELSIF bFiberOn = TRUE AND bManualChop = TRUE THEN
		iFiberPres :=32000*iFiberScale/100;
		ELSE iFiberPres :=0;
END_IF
IF bFiberOn = FALSE THEN
	iFiberPres :=0;
END_IF
IF bManualChop = TRUE AND bFiberOn= TRUE THEN
	iFiberPres :=32000*iFiberScale/100;
END_IF

END_PROGRAM

// ---- Machine System/PRGs/CAM_CNC/Gun/myPressure.TcPOU
PROGRAM myPressure
VAR
	iResinP : UINT;
	iAcetoneP : UINT;
	iGunMacsP AT %I* : UINT;
	myAir :INT;
END_VAR



//resin and MEK pump pressure


//acetone pump pressure


//itv for chopper (may add chopper to spindle on hmi interface to adjust the itv value


//gun mac pressure

END_PROGRAM

// ---- Machine System/PRGs/Rib Machine/START_STOP_1.TcPOU
PROGRAM START_STOP_1
VAR
	START_TIMER : TON;
	START_TIMER_ELAPSED: TIME;
	START_TIMER_DONE : BOOL; 
	START_PB AT %I*:BOOL;
	STOP_PB AT %I*:BOOL;
	START_REQUEST:BOOL;
	STOP_REQUEST:BOOL;


END_VAR
VAR // added by the converter: edge detectors and wires of the graphical bodies
    _rt1 : R_TRIG;
END_VAR

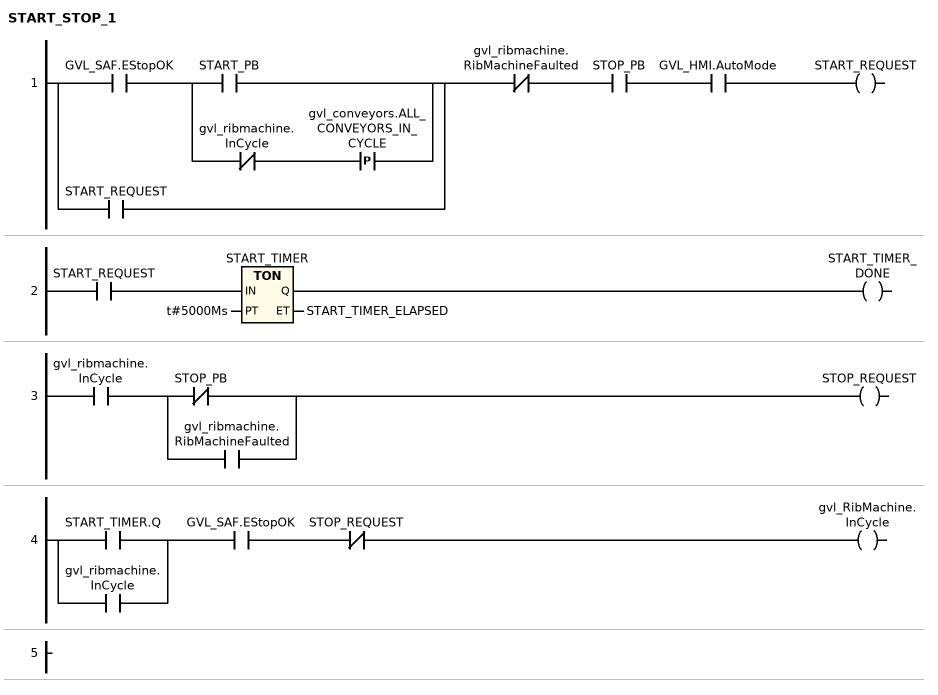
// NETWORK 1
_rt1(CLK := gvl_conveyors.ALL_CONVEYORS_IN_CYCLE);
START_REQUEST := (GVL_SAF.EStopOK AND (START_PB OR NOT gvl_ribmachine.InCycle AND _rt1.Q) OR START_REQUEST) AND NOT gvl_ribmachine.RibMachineFaulted AND STOP_PB AND GVL_HMI.AutoMode;

// NETWORK 2
START_TIMER(IN := START_REQUEST, PT := t#5000Ms, ET => START_TIMER_ELAPSED); // TON
START_TIMER_DONE := START_TIMER.Q;

// NETWORK 3
STOP_REQUEST := gvl_ribmachine.InCycle AND (NOT STOP_PB OR gvl_ribmachine.RibMachineFaulted);

// NETWORK 4
gvl_RibMachine.InCycle := (START_TIMER.Q OR gvl_ribmachine.InCycle) AND GVL_SAF.EStopOK AND NOT STOP_REQUEST;

// NETWORK 5

END_PROGRAM

// ---- Machine System/PRGs/SprayRibRollCureSequencerSD1.TcPOU
PROGRAM SprayRibRollCureSequencerSD1
VAR
	bInit : BOOL; // This sequence has been initialized.
	
	bLoading    : BOOL; // The sequence is loading tools into the bogie arms
	
	bSpraying   : BOOL; // The sequence is spraying the tools
	bRolling    : BOOL; // The sequence is rolling the tools
	bRibbing    : BOOL; // The sequence is ribbing the tools
	bCuring     : BOOL; // The sequence is curing the tools
	
	bUnloading  : BOOL; // The sequence is unloading tools from the bogie arms
	bTraversing : BOOL; // The arms are jogging.
	
	bAbleToUnload : BOOL; // TRUE when there are no part(s) blocking unload position | FALSE when there are part(s) blocking the unload position
	
END_VAR
(*
	THIS CURRENT VERSION OF THE SEQUENCER IS JUST FOR A DEMO DRY RUN WITH WX2.

	Definitions :
	Loading) We are 'Loading' until the arms have picked up the tool, and then moved them into the correct angle for spraying.
	Spraying) We are Spraying until the .NC file that is being ran by the CNC program has completed.
	Rolling) We are 'Rolling' until the .NC file that is being ran by the CNC program has completed.
	Ribbing) We are 'Ribbing' until the .NC file that is being ran by teh CNC program has competed.
	Curing) We are 'Curing' once we get into the cure position (rotation and horizontal positions) until the 'Curing timer' = 0;
	Traversing) we are considered 'moving' until we are in both the correct position with the SD jog and bogie arm rotation.
	Unloading) We are unloading until the tool has been set down, unclamped, and the arms have moved into their traverse position.
	
*)

	// These variables are for error related machine states.
VAR
	bError : BOOL;
END_VAR

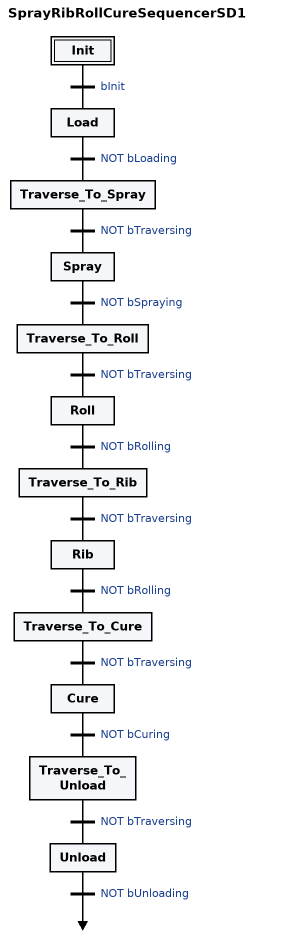
INITIAL_STEP Init:
END_STEP
TRANSITION FROM Init TO Load
    := bInit;
END_TRANSITION
STEP Load:
END_STEP
TRANSITION FROM Load TO Traverse_To_Spray
    := NOT bLoading;
END_TRANSITION
STEP Traverse_To_Spray:
END_STEP
TRANSITION FROM Traverse_To_Spray TO Spray
    := NOT bTraversing;
END_TRANSITION
STEP Spray:
END_STEP
TRANSITION FROM Spray TO Traverse_To_Roll
    := NOT bSpraying;
END_TRANSITION
STEP Traverse_To_Roll:
END_STEP
TRANSITION FROM Traverse_To_Roll TO Roll
    := NOT bTraversing;
END_TRANSITION
STEP Roll:
END_STEP
TRANSITION FROM Roll TO Traverse_To_Rib
    := NOT bRolling;
END_TRANSITION
STEP Traverse_To_Rib:
END_STEP
TRANSITION FROM Traverse_To_Rib TO Rib
    := NOT bTraversing;
END_TRANSITION
STEP Rib:
END_STEP
TRANSITION FROM Rib TO Traverse_To_Cure
    := NOT bRolling;
END_TRANSITION
STEP Traverse_To_Cure:
END_STEP
TRANSITION FROM Traverse_To_Cure TO Cure
    := NOT bTraversing;
END_TRANSITION
STEP Cure:
END_STEP
TRANSITION FROM Cure TO Traverse_To_Unload
    := NOT bCuring;
END_TRANSITION
STEP Traverse_To_Unload:
END_STEP
TRANSITION FROM Traverse_To_Unload TO Unload
    := NOT bTraversing;
END_TRANSITION
STEP Unload:
END_STEP
TRANSITION FROM Unload TO _
    := NOT bUnloading;
END_TRANSITION

END_PROGRAM

// ---- Messages/myMESSAGES.TcPOU
PROGRAM myMESSAGES
VAR
	i : INT;
END_VAR

MSG_ALARM_List[1] := NOT bEstopPB;
MSG_ALARM_List[2] := bProbeLowBattery;
MSG_ALARM_List[3] := bProbeError;
MSG_ALARM_List[4] := NOT bAtcVfdFaultedState;
MSG_ALARM_List[5] := NOT bDriveFaultSpindle;
MSG_ALARM_List[6] := NOT bDriveFaultAtcCarrousel;
MSG_ALARM_List[7] := NOT bDriveFaultAtcArm;
MSG_ALARM_List[8] := NOT bAtcArmTorqueSw ;
MSG_ALARM_List[9] := FALSE;(*NOT (gpAx[0]^.lr_state.homing_done_r AND gpAx[1]^.lr_state.homing_done_r AND gpAx[2]^.lr_state.homing_done_r AND axAtcCarrousel.Status.Homed AND axAtcArm.Status.Homed);
	IF CNCSystem.Channel[0].Mode.Auto OR CNCSystem.Channel[0].Mode.MDI THEN
		IF MSG_ALARM_List[9] THEN
			PLCMachineMode[0].Manual := TRUE;
		END_IF
	END_IF*)

//MSG_ALARM_List[10] := True; // send msg that there is no pressure value with M10 pipe clamp or it is out of range
//MSG_ALARM_List[11] := true; // send msg that the tool in spindle is unknown
//MSG_ALARM_List[12] := TRUE; // send msg that drawbar switches are not adjusted properly
//MSG_ALARM_List[13] := TRUE;// send msg that all axis are not homed
//MSG_ALARM_List[14] := TRUE;// message = AtcCarousel not in position
//MSG_ALARM_List[15] := TRUE;// message = AtcArm not in position
//MSG_ALARM_List[16] := TRUE;// send msg carriage did not get to fwd limit in time
//MSG_ALARM_List[17] := TRUE;// message = Atc Arm not clear to move
//MSG_ALARM_List[18] := TRUE;//message = Carousel not clear to move
//MSG_ALARM_List[19] := TRUE;//message = Carriage not clear to move
//MSG_ALARM_List[20] := TRUE; // send msg carriage did not get to fwd limit in time
//MSG_ALARM_List[21] := TRUE; // send msg that there is no tool detected in new tool pocket
//MSG_ALARM_List[22] := TRUE; // send msg that drawbar sensor for tool loaded is missing
//MSG_ALARM_List[23] := TRUE; // send msg that axes need to be moved off of home switches before homing
MSG_ALARM_List[24] := wHorzDriveStatusWord.3;
MSG_ALARM_List[25] := wVertDriveStatusWord.3;
MSG_ALARM_List[26] := rActualCounterBalancePressure < 68; // Counter balance pressure too low
MSG_ALARM_List[27] := rActualCounterBalancePressure > 72; // Counter balance pressure too high
MSG_ALARM_List[28] := NOT bAtcManualToolReleaseSw; // manual tool release handle is not retracted
IF bResetPB THEN
	FOR i := 1 TO 50 BY 1 DO
		MSG_ALARM_List[i] := FALSE;
	END_FOR
END_IF

END_PROGRAM

// ---- Messages/myPlcMessages.TcPOU
PROGRAM myPlcMessages
VAR
	nAirPressureValue :int;
	nCycleCounts: INT;
END_VAR

HmiMessages[0] := 'Air Pressure';
HmiMessagesValues[0] := INT_TO_STRING(nAirPressureValue);
IF nAirPressureValue < 120 THEN
	HmiMessagesColor[0] := 16#FFFF0000; // RED box
ELSE
	HmiMessagesColor[0] := 0;
END_IF

HmiMessages[1] := 'Cycle Counter';
HmiMessagesValues[1] := INT_TO_STRING(nCycleCounts);

END_PROGRAM

// ---- Machine System/FBs/CP/ClampCPLinPPR.TcPOU
FUNCTION_BLOCK ClampCPLinPPR EXTENDS ClearpathPositionLinPPR
VAR_INPUT
	PartPresentHi AT %I* : BOOL;
	PartPresentLo AT %I* : BOOL;
END_VAR
VAR_OUTPUT
	PartPresent_PO	: BOOL;
	PartPresent_VO	: BOOL;
	HomeStatusMsg_VO : string;	
END_VAR
VAR
	ClampHomeCase : INT;
END_VAR


IF Mode_PI =1 THEN //autohoming in automode
	CASE ClampHomeCase OF
		0:  
			IF Out.Homed_PO =0 AND PartPresentHi =0 AND PartPresentLo=0 THEN
			 ClampHomeCase :=20;
			END_IF
			IF Out.Homed_PO =0 AND PartPresentHi =1 AND PartPresentLo =1 THEN
			//Part in clamp set home at xx distance and set home
			ClampHomeCase:=10;
			END_IF
		10: //use psudeo home against part pipes
			Out.Homed_PO:=1;
			HomeCase:=0;
			Out.DistancePos_PO:=120;
			pulsecount :=120; //dis *2 (2 ppr per dis on base)
			expectedPulse :=120; //dis *2 (2 ppr per dis on base)
			Out.ExpDistancePos_PO :=120;
			ClampHomeCase:=0;
		20: //Use clamp home start
			bHomeStart_PI :=1;
			IF Out.Homed_PO THEN 
				ClampHomeCase:=0;
			END_IF
		
		30: //only one partpresnt is on.  Home, exetend and try again or flip error code
			ClampHomeCase:=0;
			HomeStatusMsg_VO:='homing not possible only one part present sensor is on. Manual reset req';
		
	END_CASE
	
END_IF

END_FUNCTION_BLOCK

// ---- Machine System/FBs/CP/ClearpathPositionLinPPR.TcPOU
FUNCTION_BLOCK ClearpathPositionLinPPR //please check comments inside FB to determine clearpath settings before use
VAR_INPUT
	
	//PI (Program Inputs)
		bHomeStart_PI				: BOOL;		//begin Homing sequence
		PowerOn_PI					: BOOL;		//enable motor command from program
		Stop_PI						: BOOL;		//stop command from program
		DistancePosReq_PI			: REAL;		//distanct position request from the program (input in absolute position and valid after homing)
		ManualMove_PI				: BOOL;		//Call manual move method if true
		Mode_PI						: INT;		//0:noMode, 1:Auto, 2:Manual
		bMove_PI					: BOOL;		//begin absolute move
		VEReq :LREAL;
	//VI (visualization input/hmi input)
		Reset_VI			: BOOL;		//reset button	
		DisReq_VI			: REAL;		//Disreq for absolute auto move	
		JogExecute_VI		: BOOL;		//Call manual move method if true
		SuperJogExecute_VI	: Bool;		//call super manual move method if true
		SuperJogMode_VI		: BOOL;		//Super Mode on if true (changes Jog method) use for overtravel or not homed be Cautious
		JogSlow_VI			: BOOL;		//slow manual move
		CW_VI				: BOOL;		//Set Direction for requested move (does not apply to absolute move) True = Clockwise
	//CI (configuration input)
		IN							: LinPPR_CI;
END_VAR
VAR_OUTPUT
	//Outputs
		Out						: LinPPR_Out;
END_VAR
VAR
	AltSpeedCase		: INT;		//case tracker altspeed()
	AltSpeedReq			: BOOL;		//turn altspeed method on
	ResetCase			: INT; 		//makes a reset instead of an alt speed request (delays the turning off of reset)
	HomeCase			: INT;		//case tracker home()
	JogCase				: INT;		//case tracker Jog()
	SuperJogCase		: INT;		//case tracker SuperJog()
	DisToGoCase			: INT;		//case tracker MoveABSLin() for pulse train que
	PositionCase		: INT;
	SWLimitStatus		: BOOL;		//Used to check if currently within software limits
	testBOol			: BOOL;		//tester
	error				: INT;		//5: increment error
	PulsesEnabled		: BOOL;		//enable absolute move method to command pulses
	busy				: BOOL;		//move in progress
	MoveComplete		: BOOL;		//all ppr accounted for after move command
	PulseCount			: INT;		//current Pulse Count
	expectedPulse		: INT;		//expected pulses from commanded movements at set PPR
	HomeTrig			: R_trig;	//trigger position capture when homing ends
	ATrig				: R_trig;	//counter/trigger to track how many increments of a output have been commanded
	pulseCounter		: r_trig;
	JogRTrig			: R_Trig;	//jog execute trigger
	JogFTrig			: F_Trig;	//Jog Cancel Trigger
	bMoveTrig			: r_trig;
	JogReset			: bool;
	ASG					: BOOL;		//all systems go clearpath (if using asg)
	Cancelled			: BOOL;		//move was cancelled requires reset
	CW					: BOOL; 	//direction of motor rotation: CW is true;  CCW is false;
	DistanceToGo		: REAL;		//difference in distance from current position and requested position.  used to determine linear direction
	isConfigured		: BOOL;		//turns on or off the configuration settings method so it only runs on first scan
	DistPerMRev 		: INT;
	testlimit			: INT;
	testR				: INT;
	DisPerPulse			: INT;		//distance per pulse based on configuration inputs
	PulsesToSend		: INT;		//Pulses to send for Absolute move
	CWABS				: BOOL;		//Direction for abs Move [Check against pulse wrong dir]
	testpulsecnt		: INT;		//testing flot vs int
	PulseQueSet			: BOOL;		//start pulses for move
	PulseQue			: int;		//int counter to hold the number of pulses left to send
	LastDistancePosReq	: real;
	//FI (Field Inputs)

	HLFB_FI	 		AT %I*	: BOOL;		// high level feedback sensors
	bInputBCom_FI	AT %I*	: BOOL;		// check sum for inputb signal	(double check that direction is actually signaled to motor)
	
	//Linear Homing Variables
	bHigh_FI		AT %I*	: BOOL;
	bLow_FI			AT %I*	: BOOL;
	bHome_FI		AT %I*	: BOOL;
	
	//FO (Field Outputs)
	HLFB24V_FO 			AT %Q*	: BOOL :=1;	//high level feedback 24v power if needed to used el2008 //default set to true so that hlfb is fucntional
	EnableOut_FO 		AT %Q* 	: BOOL; 	//enables the clearpath motor
	InputAOut_FO 		AT %Q* 	: BOOL; 	//input A of clearpath motor, output from plc
	InputBOut_FO 		AT %Q* 	: BOOL; 	//input B of clearpath motor, output from plc
	
END_VAR
VAR RETAIN 
	
	
END_VAR

VAR_IN_OUT

END_VAR

(* Checck clearpath settings before use*)
	(* Check the input filter setting for inputA and inputB.   Also check PPR setting, CntsPerPulse, HLFBsetting, and The type of axis,  
		Place clearpath in correct mode of operation Mode for this FB is position 
		Check what Homing setting is used on the clearpath motor	
		check to make sure that the resolution of movement commands matches gearbox compatibiltiy, and plc scan compatability
		
		How the FB works Details:
			1st scan sets configuration using MechDrive_CI()
			Each scan CP motor direction is set based off CW variable
			LocatePosition() drives limit switches and rotary cam limit quadrants
			Pulses are counted using ppr() to move with hlfb rising trig counter.  Expected pulses are tracked with inputA_FO rising trig
			Enable checks for enable signal, cancelled state, and stop_PI state before turning on motor or disenable
			reset: cp motors require an enable off to reset after ac loss...ie estop w/contactor.  it also resets cancelled bit and busy bit (requires reset_vi to run)
			
			Moves are called using homing sequence, Absolute movement, or with manual movement and all require homing.
			after homing absolute movement within software limit_CI is available or manual jog.  Manual jog is set to single pulse method by default
			After Homing Position is tracked using 'DistancePos_PO'
			ABsolute move chains clearpath pulses together to create a smooth motion profile. 
				Pulses sent are tracked against 'DistancePosReq_PI' and 'DistancePos_PO'  When expected pulses are within range of requested position then 'pulsecount' is reset
	*)
(*configruation input setting*)
IF isConfigured = 0 THEN MechDrive_CI();	END_IF	//run once to set configuration on init

//Pin outs Clockwise (CW) or Counter Clockwise (CCW)
IF CW THEN	InputBOut_FO := 1;	ELSE InputBOut_FO := 0; 	END_IF //sets direction of movement at motor - check this (add bcom direction pin check)
LocatePosition();				//rotary position of the cam wheel  //also includes a double sensor check for SensorCheck_PO  //Also locates position for linear system for limit sensors //Limits
//Triggers
	pulseCounter(clk:=HLFB_FI);		//high Level feedback counter based off direction
	HomeTrig(clk:=Out.Homed_PO);		//used in ppr() to set pulses to zero after homing
	ATrig (clk:=InputAOut_FO);		//counts pulses sent to motor (clearpath should move based on InputA Rising Trig (check settings in CP to be sure - options are for rising or falling trig)
	JogRTrig(CLK:=JogExecute_VI);	//Starts Jog()
	JogFTrig(CLK:=JogExecute_VI);	//Cancels Jog() movement
	bMoveTrig(Clk:=bmove_PI,); 		//confirms that move has triggered and then can check MDI MCode Req Pos
IF Mode_PI =2 THEN
	IF SuperJogMode_VI =0 THEN
		Jog(); ELSE SuperJog();
	END_IF
	Out.ModeMsg_VO :='Manual Mode Engaged';
END_IF
IF Mode_PI =1 THEN
	DistancePosReq_PI:=DisReq_vi;
	MoveAbsLin();
END_IF
PPR();							//tracking of the Pulses per revolution if using ppr (default for most use cases)
Home();
//moved movedone into movement manula call and abs move call
MoveDone();						//check if movement is complete (will either check pulses against expected pulses or will check for asg
Enable();						//check for motor enable status and try to enable the motor if PowerOn_PI is true
Reset();						//if reset button turn power off, reset cancelled, and reset busy
IF stop_PI THEN CancelMove(); END_IF	//This requires a reset afterwards to move again

METHOD PUBLIC AltSpeed : BOOL
VAR_INPUT
END_VAR
(*clearpath requires at least a 20ms delay where the enable signal is pulsed off to realize alternate speed *)

//start
CASE AltSpeedCase OF
	0:
		altspeedcase :=10;
	10:
		EnableOut_FO :=1 ;
		AltSpeedCase :=20;
	20:
		EnableOut_FO :=1;
		AltSpeedCase :=30;
	30:
		EnableOut_FO := 0 ;
		AltSpeedCase :=40;
	40:
		EnableOut_FO := 0;
		AltSpeedCase := 50;
	50:
		EnableOut_FO := 0 ;
		AltSpeedCase := 60;
	60:	
		EnableOut_FO := 1 ;
		//Look for 'AltSpeedCase' to be set to '0' in the call function
	
	90: //error or message
END_CASE
END_METHOD

METHOD PUBLIC CancelMove : BOOL
VAR_INPUT
END_VAR
EnableOut_FO 	:= 0;		//only way to clear out overstacked increment calls is to turn enable off and then on
//PowerOn_PI		:=0;	//turn off power on [this is a program input and can't be turned off here] check this to see if still needed[was affecting homecase]
Cancelled	:=1;	//cancelled move needs to be reset
expectedpulse := pulsecount;	//resets expected pulse after an estop or limit switch event
Out.DistancePos_PO := Pulsecount/2; //PPRset_CI*1	//resets distance counter to position after a cancelled move
Out.ExpDistancePos_PO := PulseCount/2; //change distancePOs_PO to float if needed
DisToGoCase :=0;
PulsesToSend :=0;
AltSpeedReq :=0;	//clear alt speed mode	
AltSpeedCase :=0;	
InputAOut_FO :=0;
// message (move was canceled)
END_METHOD

METHOD PUBLIC DisToGo : BOOL
VAR_INPUT
END_VAR
IF Out.Homed_PO THEN
	IF DistancePosReq_PI > Out.ExpDistancePos_PO THEN 
		CW := 1;	//move CW to reach req position
	END_IF
	IF DistancePosReq_PI < Out.ExpDistancePos_PO THEN
		CW :=0;	//Move CCW to reach req position
	END_IF
(*	IF PulseQue >0 THEN 
		PulsesEnabled:=1;
		ELSE PulsesEnabled :=0; 
	END_IF *)
	
	IF DistancePosReq_PI = Out.ExpDistancePos_PO THEN 
		PulsesEnabled :=0;
		CW := CW;
		ELSE
			PulsesEnabled := 1;
	END_IF

	ELSE
	//check this (is the homed block required?)
	//Message that Movement cant be made until homing has occured or use manual mode	
	
END_IF

(*
if pulseQue is > 0 then PulseEnabled;
*)
END_METHOD

METHOD PUBLIC Enable : BOOL 	//attempts to enable the motor based on stop_PI, Cancelled, and PowerOn_PI
VAR_INPUT
END_VAR
IF Stop_PI =0 AND cancelled =0 AND PowerOn_PI =1 AND ResetCase=0 THEN
	EnableOut_FO :=1;
	IF altSpeedReq THEN
		AltSpeed();				//calls altspeed to cycle thru if homing or manual mode requests a slower mode
	END_IF
	ELSE EnableOut_FO :=0;	//message to say stop is on (check this)
END_IF


//power on

//check if asg

//if no asg power off and repeat
END_METHOD

METHOD PUBLIC Error : BOOL
VAR_INPUT
END_VAR
// if hlfb pulses do not move in set timeframe after movement call then call error for motor
END_METHOD

METHOD PUBLIC Home : BOOL
VAR_INPUT
END_VAR
//limit switch and home switch configuration
IF IN.HomingSet_CI = 2 THEN //homing sensor not used - home to low sensor
bHome_FI := bLow_FI; 
//message homing sensor not used
END_IF
IF IN.HomingSet_CI = 3 THEN //homing sensor not used - home to Hi sensor
	bHome_FI := bHigh_FI; 
	//message homing sensor not used
END_IF
//error catch for if InputBout wire fails and ends up homing unknown direction repeatedly
IF PowerOn_PI = 0 THEN HomeCase :=0; END_IF
IF Stop_PI = 1 THEN HomeCase := 0; END_IF
//check the InputBOut com using EL1008 input channel to determine that the pulse did work
//message
IF bhomestart_PI = 1 THEN HomeCase :=0; AltSpeedReq := 1; AltSpeedCase:=0; END_IF
CASE HomeCase OF
	0://set pulses equal so that movement can begin and check direction
		IF bHomeStart_PI =1 AND Stop_PI = 0  THEN
			HomeCase := 10;
			bhomeStart_PI :=0;
			AltSpeedReq := 1;				//set slow mode and alternate speed in clearpath
			//AltSpeedCase := 0;			//may need this to start slow speed
			ExpectedPulse := PulseCount;	//Make movement available no matter the pulse count discrepancy
			InputAOut_FO :=0;
			Out.Homed_PO :=0;
		END_IF
	(*5:	
		IF Stop_PI = 0  THEN
			HomeCase := 10;
			bhomeStart_PI :=0;
			AltSpeedReq := 1;				//set slow mode and alternate speed in clearpath
			AltSpeedCase := 0;
			ExpectedPulse := PulseCount;	//Make movement available no matter the pulse count discrepancy
			Homed_PO :=0;
		END_IF*)
		
	10:// homing sequence
		IF  Stop_PI = 0  THEN
			Out.Homed_PO :=0;
			//check this: reseting expected to match pulse count so that homeing will start if there is a mismatch
			//decide homing direction and homing method //make flag large enough to hit home switch and the limit switch
			IF IN.Limit_NC_NO_CI =0 THEN	//NC switch configuration
				IF bHigh_FI =1 AND bLow_FI =1 THEN	//using normally closed sensor (flag is not on either limit switch)
					IF IN.HomingSet_CI =2 THEN cw := 0; ELSIF IN.HomingSet_CI =3 THEN cw :=1; END_IF //go to high or low first if no limit switch tripped
				END_IF
			ELSE	//NO switch Configuration
				IF bHigh_FI =0 AND bLow_FI =0 THEN	//using normally closed sensor (flag is not on either limit switch)
					IF IN.HomingSet_CI =2 THEN cw := 0; ELSIF IN.HomingSet_CI =3 THEN cw :=1; END_IF //go to high or low first if no limit switch tripped
				END_IF
			END_IF
			//if inputA is hi then turn off (takes 2 cycles to output an increment at cp motor)
				(*if pulses expected = pulse count then do the next move *)
			IF AltSpeedCase = 60 THEN SendPulse(); END_IF
			IF IN.Limit_NC_NO_CI =0 THEN	//NC switch configuration
				IF bHome_FI =0 THEN //use nc switch for sensor [at home position]
					bHomeStart_PI :=0;
					Cancelmove();
					HomeCase := 20;
				END_IF
				ELSE				//NO switch configuration
				IF bHome_FI =1 THEN //use no switch for sensor [at home position]
				bHomeStart_PI :=0;
				Cancelmove();
				HomeCase := 20;
			END_IF	
			END_IF
			(*check this - add in an extra cycle before setting home that moves away from the 
				homed spot in same direction to confirm trigger positino comes on same side of sensor each time*)
		END_IF
	20:	//extra scan before homed
		HomeCase :=50;	//this scan is required to allow for a cancelled move reset after homing
	
	50://after homing reset motor and cancelled bit
		
			Out.Homed_PO := 1;
			//cancelled :=0;	//resets motor after initial homing
			pulsecount :=0;
			expectedPulse :=0;
			Out.DistancePos_PO :=0;
			Out.ExpDistancePos_PO :=0;
			testbool := TRUE;
			HomeCase := 0;	//back to the start
	90://reset to default or?
	
END_CASE
END_METHOD

METHOD PUBLIC InLimits : BOOL
VAR_INPUT
	Req	: REAL;	//reqested degree or position from abs move to be evaluated for limits
END_VAR
//only valid after homing
InLimits := TRUE;
IF IN.SWLimit_Hi_CI <=0 OR IN.SWLimit_Lo_CI >=0 THEN		//check this (may need to have a neg hi at some point)
	//message to say no limits are set
	InLimits :=FALSE;	
END_IF
IF Req <= IN.SWLimit_Hi_CI AND Req >= IN.SWLimit_Lo_CI THEN
	InLimits := TRUE;
	ELSE
		InLimits :=FALSE;
END_IF
END_METHOD

METHOD PUBLIC Jog : BOOL
VAR_INPUT
END_VAR

//add software limits check this
CASE JogCase OF 
	0:	//Main Jog Sequence [Also stops movement]
		IF JogSlow_VI THEN AltspeedReq :=1; ELSE AltSpeedReq :=0;   END_IF
			
		IF JogExecute_VI AND Out.Homed_PO =1  THEN	//if last move is done then allow for manual increment also required to be at home //check sensor check
			IF IN.Limit_NC_NO_CI = 0 THEN	//NC limit switch configuration
				IF bHigh_FI AND bLow_FI THEN //set direction via hmi unless on a limit switch then default to locateposition()
					IF CW_VI = 1 	THEN	CW := 1; 	ELSE CW:=0; 	END_IF
					IF bhigh_fI = 0	THEN 	CW:=0; 		END_IF
					IF bLow_FI = 0 	THEN 	CW:=1; 		END_IF
				END_IF
				ELSE	//NO limit switch configuration
					IF bHigh_FI =0 AND bLow_FI  = 0 THEN //set direction via hmi unless on a limit switch then default to locateposition()
					IF CW_VI = 1 	THEN	CW := 1; 	ELSE CW:=0; 	END_IF
					IF bhigh_fI = 1	THEN 	CW:=0; 		END_IF
					IF bLow_FI = 1 	THEN 	CW:=1; 		END_IF
				END_IF
			END_IF
			IF AltspeedReq THEN			// slowjog if altspeed is requested and wait for case 60
				IF AltspeedCase = 60 THEN
					SendPulse();
					
				END_IF
				ELSE
					SendPulse();		//send pulse for reg speed jog
			END_IF
			ELSE
				IF	JogExecute_VI  = FALSE THEN		
					CancelMove();
					JogCase :=10;
				END_IF
		END_IF
	10:	//go for auto jog reset
		IF cancelled THEN jogCase :=20; END_IF
	20: //auto Reset cycle
		IF InLimits(Out.DistancePos_PO) THEN JogCase :=30; ELSE JogCase:=95;  END_IF
	30: JogCase :=31; //10 scan delay
	31: JogCase :=32;
	32:	JogCase :=33;
	33: JogCase :=34;
	34: JogCase :=35;
	35: JogCase :=36;
	36: JogCase :=37;
	37: JogCase := 38;
	38: JogCase := 39;
	39: JogCase :=40;
	40: //send auto jog reset
		JogReset := 1;
		JogCase :=50;
	50: //wait for jog to reset
		IF JogReset=0 THEN JogCase :=90; END_IF 
	60:
	70:
	80:
	90: IF JogExecute_VI =TRUE THEN JogCase :=0; END_IF
	95: //outside of limits	
		if Reset_VI then JogCase:=90; End_if //no autoreset if outside limits
	
END_CASE
END_METHOD

METHOD PUBLIC LocatePosition : Bool //determines if sensorcheck is on and working.  Enables movement
VAR_INPUT
END_VAR

// Linear axis limit sensors
(*		bHigh_FI		AT %I*	: 	BOOL;
		bLow_FI			AT %I*	: 	BOOL;
		bHome_FI		AT %I*	: 	BOOL;*)
//NC limit sensor configuration
IF IN.Limit_NC_NO_CI = 0 THEN
	IF bHigh_FI =0 AND bInputBCom_FI =1 AND CW = 1 THEN	//use normally closed sensor and check inputb(-) [applies when trying to move past limit]
		cancelmove();
		CW := 0;	//require next move to be in Neg direction or CCW  //manual move will need to be used to get off limit switch check this
		//message saying that high limit as been exceeded or inputbcom is not connected
		Out.ErrorMsg_VO := 'High Limit reached, reset and move away from limit';
	END_IF
	IF bLow_FI =0 AND bInputBCom_FI = 0 AND CW =0 THEN	//use normally closed sensor and check inputb(-) [applies when trying to move past limit]
		cancelmove();
		CW :=1;	//require next move to be in Neg direction or CCW //manual move will need to be used to get off limit switch check this
		//message saying that Low limit as been exceeded or inputbcom is not connected
		Out.ErrorMsg_VO := 'Low Limit reached, reset and move away from limit';
	END_IF
ELSE
	//NO limit sensor configuration
	//additional option to use a N/O sensor if desired....not suggested
	IF bHigh_FI =1 AND bInputBCom_FI =1 AND CW = 1 THEN	//use normally closed sensor and check inputb(-) [applies when trying to move past limit]
		cancelmove();
		CW := 0;	//require next move to be in Neg direction or CCW  //manual move will need to be used to get off limit switch check this
		//message saying that high limit as been exceeded or inputbcom is not connected
		Out.ErrorMsg_VO := 'High Limit reached, reset and move away from limit';
	END_IF
	IF bLow_FI =1 AND bInputBCom_FI = 0 AND CW =0 THEN	//use normally closed sensor and check inputb(-) [applies when trying to move past limit]
		cancelmove();
		CW :=1;	//require next move to be in Neg direction or CCW //manual move will need to be used to get off limit switch check this
		//message saying that Low limit as been exceeded or inputbcom is not connected
		Out.ErrorMsg_VO := 'Low Limit reached, reset and move away from limit';
	END_IF
END_IF
Out.LastDistancePos_PO := Out.DistancePos_PO;
END_METHOD

METHOD PUBLIC MechDrive_CI : BOOL
VAR_INPUT
END_VAR
// 0: motor only(rot), 1: Motor and gear(rot), 2: Motor w/gear and screw(lin), 3: Motor w/screw only(lin), 4: Motor w/gear and pulley(lin),  5: Motor w/pulley(lin), 8: bypass mode
(*		DistPerMRev_CI		:	INT;	//distance traveled per rev		(Calculate your own pitch and lead w/gearbox combo must set MechDriveType_CI to 8 to bypass internal calc)
		DegPerMRev_CI		:	INT;	//distance traveled per rev		(Calculate your own pitch and lead w/gearbox combo must set MechDriveType_CI to 8 to bypass internal calc)
		DisPerFPulley_CI	:	INT;	//distance traveled per rev of final pulley (mm)
		GearRatio_CI		:	INT;	// GearRatio motor to moving part (XX:1) (gearbox and lead included in calc for vert axis) (use this for gearbox and pulleys as well)
		Lead_CI				:	INT;	// Lead of Screw if used (mm)			 (gearbox and lead included in calc for vert axis)	
*)

IF IN.MechDriveType_CI = 2 THEN	//2: Motor w/gear and screw(lin)
	DistPerMRev := IN.Lead_CI/IN.GearRatio_CI;	//driven mech ex 4mm/40 = .1mm per rev
	Out.MechTypeMsg_VO := 'Motor w/gear ratio and screw - no Degrees available [no rotary by default]';
	IF IN.GearRatio_CI <=0 OR IN.Lead_CI <=0 THEN
		isconfigured :=0;
		Out.MechTypeMsg_VO := 'GearRatio_CI or Lead_CI not configured please configure to continue';
	END_IF
END_IF

IF IN.MechDriveType_CI = 3 THEN	//3: Motor w/screw only(lin)
	DistPerMRev := IN.Lead_CI;		//driven mech ex 4mm = 4mm per rev
	Out.MechTypeMsg_VO := 'Motor w/screw - no Degrees available [no rotary by default]';
	IF IN.Lead_CI <=0 THEN
		isconfigured :=0;
		Out.MechTypeMsg_VO := 'Lead_CI not configured please configure to continue';
	END_IF
END_IF

IF IN.MechDriveType_CI = 4 THEN	//4: Motor w/gear and pulley(lin),
	DistPerMRev := IN.DisPerFPulley_CI/IN.GearRatio_CI;	//pulley circumference (20t at10 ~ 200mm per fin rev/gear ratio (40) = 5mm/motor rev
	Out.MechTypeMsg_VO := 'Motor w/gear ratio and pulley [no Degree used by default (linear pulley drive) if a rotary either use bypass or use type 1 and include pulley in gear ratio]';
	IF IN.GearRatio_CI <=0 OR IN.DisPerFPulley_CI <=0 THEN
		isconfigured :=0;
		Out.MechTypeMsg_VO := 'GearRatio_CI or DisPerFPulley_CI not configured please configure to continue';
	END_IF
END_IF

IF IN.MechDriveType_CI = 5 THEN	//5: Motor w/pulley(lin);
	DistPerMRev := IN.DisPerFPulley_CI;	//pulley circumference (20t at10 ~ 200mm per fin rev/gear ratio (40) = 5mm/motor rev
	Out.MechTypeMsg_VO := 'Motor w/pulley [no Degree used by default (linear pulley drive) if a rotary either use bypass or use type 1 and include pulley in gear ratio]';
	IF IN.DisPerFPulley_CI <=0 THEN
		isconfigured :=0;
		Out.MechTypeMsg_VO := 'DisPerFPulley_CI not configured please configure to continue';
	END_IF
END_IF

IF IN.MechDriveType_CI = 8 THEN	//8 mechdrivetype is bypassed and is set via DistPerMRev_CI or DegPerMRev_CI;
	DistPerMRev := IN.DistPerMRev_CI;
	Out.MechTypeMsg_VO := 'MechDriveType is bypassed - use DegPerMRev_CI or DistPerMRev_CI';
	IF IN.DistPerMRev_CI <=0  THEN
		isconfigured :=0;
		Out.MechTypeMsg_VO := 'DistPerMRev_CI not configured please configure to continue';
	END_IF
END_IF

IF IN.InputFilter_CI <=0 THEN
	isconfigured :=0;
	Out.ConfigMSG_VO := 'Input filter not configured, please check InputFilter_CI and clearpath motor settings';
END_IF

//linear axis
DisPerPulse := (DistPerMRev*IN.cntpulseSet_CI/32000);	//check this (Likely not a correct calc)
isConfigured :=1;	//sets configuration to true so that this block only runs once
END_METHOD

METHOD PUBLIC MoveAbsLin : BOOL
VAR_INPUT
END_VAR
IF Out.Homed_PO THEN
	CASE PositionCase OF
		0:
			IF ABS(out.DistancePos_PO-LastDistancePosReq) <in.MoveABSTol_CI THEN
				Out.InTargetPosition:=1; ELSE Out.InTargetPosition :=0;
			END_IF
		10: PositionCase :=20;
		20: PositionCase :=30;
		30: PositionCase :=40;
		40: PositionCase :=50;
		50: PositionCase :=90;
		90: PositionCase :=0;
	END_CASE
	IF ABS(VEReq - Out.DistancePos_PO) < In.MoveABSTol_CI THEN
		Out.InMPos :=1; ELSE Out.InMPos:=0;
	END_IF
	IF bMoveTrig.Q THEN Out.InMPos :=0; END_IF //Set the MPos to false after move command
END_IF
IF Out.Homed_PO THEN
	CASE DisToGoCase OF
		0:	//Readyto Take Command
			IF ABS(out.DistancePos_PO-Out.ExpDistancePos_PO) < In.MoveABSTol_CI THEN Out.InPosition:=1; END_IF	//check if current pos is within tolerance
			IF Out.InPosition THEN Out.ReadyForMove_PO :=1; END_IF		//Only ready if in position
			IF Out.ReadyForMove_PO THEN
				IF bMove_PI AND InLimits(DistancePosReq_PI)THEN  //If move is within set limits and called in Prog then execute move
					DisToGoCase :=10;
					//set MCode Received Bit [Confirm acted in end case] (this is important for aux axis in cnc VE Variable calls)
				END_IF
			END_IF
		10: //check what quePulseDistance should be and set it 
			PulsesToSend := REAL_TO_INT((DistancePosReq_PI -Out.DistancePos_PO)/In.DisPerPulse_CI); //Gets number of pulses to send
			IF PulsesToSend >0 THEN CWABS:=1; ELSE CWABS:=0; END_IF 	//Sets direction for pulses (pos CW[true] neg CW[False]
			bMove_PI :=0;	//Set Req back to false
			LastDistancePosReq := DistancePosReq_PI; //set for target
			Out.ReadyForMove_PO:=0;	//set busy with abs move
			DisToGoCase :=20;
		20: //set the if homed statement for direction control set that here and move to next case
			IF CWABS THEN CW:=1; ELSE CW:=0; END_IF	//Check abs direction each round of pulse send
			IF ABS(PulsesToSend) >0 THEN 
				PulsesEnabled:=1; 
				ELSE 	PulsesEnabled :=0; 	DisToGoCase :=30; //if no more pulses move on to case 30 to check the location tolerance
			END_IF	//if any pos or neg pulses then enable pulses
			Out.InPosition :=0;
			IF PulsesEnabled =1 AND Stop_PI = 0 AND EnableOut_FO =1 AND CW = bInputBCom_FI THEN	//check for the motor being on before incrementing the distancepos from disreq	
				//if inputA is hi then turn off (takes 2 cycles to output an increment at cp motor)
				IF CW = CWABS THEN
					SendPulse();	
					ELSE //Message CW Not equal CWABS
				END_IF	
			ELSE
				error := 5; //check the inputbcom_FI feedback
			END_IF	
			//if input filter of clearpath is too high sometimes these pulses will not register (needed to maintain ability to chain moves)  Otherwise can use asg and movedone
		30: //count pulses and and when enough pulses set pulses(rounded) not enabled set moving tag
			IF ABS(out.DistancePos_PO-DistancePosReq_PI) < In.MoveABSTol_CI THEN
				Out.InPosition:=1; Out.ABSMoveMsg_VO:='In Position';//Position Reached flag and msg
				DisToGoCase := 40;
				ELSE DisToGoCase :=99; //error
			END_IF
			DisToGoCase :=40;
		40: // ready to receive next quedistance
			Out.ReadyForMove_PO :=1;
			//Send MCode confirmation to true
			DisToGoCase:=0;
	END_CASE
	(*
	IF (DistancePosReq_PI +1) >= (QuePulseDistance + Out.DistancePos_PO) AND (DistancePosReq_PI-1)  >= (QuePulseDistance + Out.DistancePos_PO)  THEN 
		PulsesEnabled :=0;
		CW := CW;
		ELSE
			PulsesEnabled := 1;
	END_IF *)
END_IF






(*
IF InLimits(DistancePosReq_PI) AND Out.Homed_PO =1 THEN //begin pulses
	IF PulsesEnabled =1 AND Stop_PI = 0 AND EnableOut_FO =1 AND CW = bInputBCom_FI THEN	//check for the motor being on before incrementing the distancepos from disreq	
		//if inputA is hi then turn off (takes 2 cycles to output an increment at cp motor)
		SendPulse();		
		ELSE
			error := 5;
		END_IF	
		//if input filter of clearpath is too high sometimes these pulses will not register (needed to maintain ability to chain moves)  Otherwise can use asg and movedone
	IF DistancePosReq_PI = Out.ExpDistancePos_PO AND MoveComplete =0 THEN 
		PulsesEnabled :=0; 
			//check this
	END_IF
ELSE
	//message not in limits	
END_IF
//add limits option here for stopping overtravel
*)
END_METHOD

METHOD PUBLIC MoveDone : BOOL
VAR_INPUT
END_VAR
//ppr setting of hlfb is required
(*movecomplete is set either when pulsecount lines up exactly or if pulseque is empty and pulsecount is within tolerance*)
	IF PulseCount = expectedPulse  THEN	// (check this - add a tolerance here)
		MoveComplete :=1; 
		MoveDone := TRUE;
		busy :=0;			//set busy to zero (these are possibly interchangable until further code added) check this
		ELSE
			MoveDone :=FALSE;
		//is movedone() not completed check this
		//Add in MOVEDONE:=True; check this
	END_IF
	//movecomplete set for absolute move ppr tolerance
	IF PulseQueSet = 1 and PulseQue = 0 AND (pulseCount >= ExpectedPulse -2 OR PulseCount <= ExpectedPulse +2) THEN
		MoveComplete :=1;
		PulseQueSet :=0;
		MoveDone := TRUE;
		Busy :=0;
		//set expected to pulscount?
		//expectedPulse := PulseCount;
	END_IF
(* set DistPos_PO based off pulsecount/pulsecountset_ci  then check expectedDistPos_PO against current *)
//check busy and move complete in asg and if busytrig then check asgtrig then set move complete
END_METHOD

METHOD PUBLIC PPR : BOOL
VAR_INPUT
END_VAR
IF PulseCounter.Q THEN
	IF InputBOut_FO =1 THEN
		PulseCount := PulseCount +1;
		ELSE
			PulseCount := PulseCount -1;
		END_IF
		//extra pulse after homing is happening here? check this
END_IF

IF ATrig.Q AND Cancelled = 0 THEN
	IF InputBOut_FO = 1 THEN 
		ExpectedPulse := ExpectedPulse + (1*IN.PPRset_CI); //does not account for cnt per rev yet
		PulsesToSend := PulsesToSend-1;			//Track ABS Pulses sent  [went pos dir so remove one from que]
		ELSE 
			ExpectedPulse := ExpectedPulse - (1*IN.PPRset_CI);
			PulsesToSend := PulsesToSend +1;	//Track ABS Pulses sent  [went neg dir so add one from que]
	END_IF
	//expectedpulse should be 32000cnts div by ppr = cnts per pulse
	//expectedPulse should be cntset_CI/320000 *(1*pprset_ci)   //30223cnts per pulse currently
END_IF
IF HomeTrig.Q THEN
	PulseCount  :=0;	//set position to zero after homing is complete
	ExpectedPulse := 0;
END_IF
IF Cancelled = 1 THEN
	expectedPulse := pulsecount;
END_IF
IF  movecomplete = 1 THEN //ppr mode
	 Out.DistancePos_PO := PulseCount/2; //change distancePOs_PO to float if needed
	 Out.ExpDistancePos_PO := PulseCount/2;
END_IF
IF  PowerOn_PI =0 THEN
	Out.DistancePos_PO := PulseCount/2; //change distancePOs_PO to float if needed	//resets DistancePos_PO if PowerOn_PI signal is interupted or turned off after if mid move
	 Out.ExpDistancePos_PO := PulseCount/2;
END_IF
Out.DistancePos_PO := PulseCount/2; //change distancePOs_PO to float if needed 
(* if expected pulses are in tolerance then pulsecount/ pprset should be used to set new dist position   
*)
END_METHOD

METHOD PUBLIC Reset : BOOL
VAR_INPUT
END_VAR
CASE ResetCase OF
	0:
		IF reset_VI =1 OR JogReset=1 THEN
			EnableOut_FO :=0;	//Turn off to reset (power on will finish reset)
			Cancelled :=0;	//reset the cancelled move bit
			busy :=0;	// check this (is reseting busy needed?)
			DisToGoCase:=0;
			ResetCase :=10;
			OUt.MechTypeMsg_VO 		:= '';		
			Out.ConfigMSG_VO		:= '';		
			Out.ErrorMsg_VO			:= '';	
			Out.Error2Msg_VO		:= '';	
			Out.Error3Msg_VO		:='';		
			Out.Error4Msg_VO 		:='';
			Out.HomeMsg_VO 			:='';				
			OUt.LimitsMsg_VO		:='';	
			Out.ABSMoveMsg_VO		:='';
			OUt.SuperJogMsg_VO		:='';
			Out.DisToGoMsg_VO		:='';
			Out.CanceledMsg_VO		:='';
			Out.ModeMsg_VO			:='';
			LastDistanceposReq := Out.DistancePos_PO;
		END_IF
	(*original section above for manual reset *)
	10: ResetCase:=20;
	20: ResetCase:=30;
	30: ResetCase:=40;
	40: ResetCase:=50;
	50: ResetCase:=60;
	60: ResetCase:=70;
	70: ResetCase:=80;
	80: ResetCase:=90;
	90: 
		ResetCase:=0;
		Reset_Vi:=0;
		JogReset:=0;
END_CASE
//reset by turning power off and then on
END_METHOD

METHOD PUBLIC SendPulse : BOOL
VAR_INPUT
END_VAR
//got rid of 'and busy =0'
IF Stop_PI = 0  AND EnableOut_FO =1 AND CW = bInputBCom_FI THEN	//check for the motor being on before incrementing the distancepos from disreq	
	IF InputAOut_FO =1  THEN 
		InputAOut_FO := 0;
	ELSE 
		IF AltSpeedReq THEN
			IF AltspeedCase =60 THEN
				InputAOut_FO :=1;		//else turn true and subtract increment counter
				AltspeedCase :=0;	//reset altspeed
				IF CW =1 THEN Out.ExpDistancePos_PO := Out.ExpDistancePos_PO +1; ELSE Out.ExpDistancePos_PO := Out.ExpDistancePos_PO - 1; END_IF
			END_IF
		ELSE
			InputAOut_FO :=1;		//else turn true and subtract increment counter
			IF CW =1 THEN Out.ExpDistancePos_PO := Out.ExpDistancePos_PO +1; ELSE Out.ExpDistancePos_PO := Out.ExpDistancePos_PO - 1; END_IF
		END_IF
		MoveComplete :=0;		//set movedone to zero and await move complete
		busy		 :=1;		//set status to busy until move complete
	END_IF	
ELSE
	//InputAOut_FO := 0;		//no trigger if stopped or direction feedback failed or if motor enable is off
	//Message Saying Move is in progress
	Error:=3;//chck inputbCom feedback
		
END_IF
END_METHOD

METHOD PUBLIC SuperJog : BOOL
VAR_INPUT
END_VAR
//using this mode will disable the two sensor safety check for manual manual mode
//homing is not required to use this and as such should be used with caution
//if not 2 sensors on and not in super mode then no movement allowed
	
	//message : at least one sensor is down please check sensors.  if movement is needed enter supermanual mode
	
//else  allow manual mode  even if not all sensors are working
	//message: you are in supermanual mode and will bypass anti collision devices.  please take caution
//add software limits check this

//add software limits check this
CASE SuperJogCase OF 
	0:	//Main Jog Sequence [Also stops movement]
		IF JogSlow_VI THEN AltspeedReq :=1; ELSE AltSpeedReq :=0;   END_IF
			
		IF SuperJogExecute_VI  THEN	//if last move is done then allow for manual increment also required to be at home //check sensor check
			(*IF IN.Limit_NC_NO_CI = 0 THEN	//NC limit switch configuration
				IF bHigh_FI AND bLow_FI THEN //set direction via hmi unless on a limit switch then default to locateposition()
					IF CW_VI = 1 	THEN	CW := 1; 	ELSE CW:=0; 	END_IF
					IF bhigh_fI = 0	THEN 	CW:=0; 		END_IF
					IF bLow_FI = 0 	THEN 	CW:=1; 		END_IF
				END_IF
				ELSE	//NO limit switch configuration
					IF bHigh_FI =0 AND bLow_FI  = 0 THEN //set direction via hmi unless on a limit switch then default to locateposition()
					IF CW_VI = 1 	THEN	CW := 1; 	ELSE CW:=0; 	END_IF
					IF bhigh_fI = 1	THEN 	CW:=0; 		END_IF
					IF bLow_FI = 1 	THEN 	CW:=1; 		END_IF
				END_IF
			END_IF*)
			IF CW_VI = 1 	THEN	CW := 1; 	ELSE CW:=0; 	END_IF
			IF AltspeedReq THEN			// slowjog if altspeed is requested and wait for case 60
				IF AltspeedCase = 60 THEN
					SendPulse();
					
				END_IF
				ELSE
					SendPulse();		//send pulse for reg speed jog
			END_IF
			ELSE
				IF	SuperJogExecute_VI  = FALSE THEN		
					CancelMove();
					SuperJogCase :=10;
				END_IF
		END_IF
	10:	//
		IF SuperJogExecute_VI =TRUE THEN SuperJogCase :=0; END_IF
		
	
END_CASE
END_METHOD

END_FUNCTION_BLOCK

// ---- Machine System/FBs/CP/ClearpathPositionLinPPR_1.TcPOU
FUNCTION_BLOCK ClearpathPositionLinPPR_1 //please check comments inside FB to determine clearpath settings before use
VAR_INPUT
	
	//PI (Program Inputs)
		IN							: LinPPR_CI;
		bHomeStart_PI				: BOOL;		//begin Homing sequence
		PowerOn_PI					: BOOL;		//enable motor command from program
		Stop_PI						: BOOL;		//stop command from program
		DistancePosReq_PI			: REAL;		//distanct position request from the program (input in absolute position and valid after homing)
		ManualMove_PI				: BOOL;		//Call manual move method if true

	//VI (visualization input/hmi input)
		Reset_VI			: BOOL;		//reset button		
		JogExecute_VI		: BOOL;		//Call manual move method if true
		SuperJogExecute_VI	: Bool;		//call super manual move method if true
		JogSlow_VI			: BOOL;		//slow manual move
		CW_VI				: BOOL;		//Set Direction for requested move (does not apply to absolute move) True = Clockwise
	//CI (configuration input)
		//PPRset_CI			: 	INT;  	//ppr setting in clearpath
		//cntPulseSet_CI		: 	INT;	//cnts per pulse clearpath setting
		//HomingSet_CI		: 	INT;	// CP_FB homing settings - 0: disabled; 1: Home to low switch 2: home to hi switch 3: home with CP Drive and asg
		//DistPerMRev_CI		:	INT;	//distance traveled per rev		(Calculate your own pitch and lead w/gearbox combo must set MechDriveType_CI to 8 to bypass internal calc)
		//DisPerFPulley_CI	:	INT;	//distance traveled per rev of final pulley (mm)
		//GearRatio_CI		:	INT;	// GearRatio motor to moving part (XX:1) (gearbox and lead included in calc for vert axis) (use this for pulleys as well)j
		//Lead_CI				:	INT;	// Lead of Screw if used (mm)			(gearbox and lead included in calc for vert axis)
		//MechDriveType_CI	:	INT;	// 0: motor only(rot), 1: Motor and gear(rot), 2: Motor w/gear and screw(lin), 3: Motor w/screw only(lin), 4: Motor w/gear and pulley(lin),  5: Motor w/pulley(lin), 8: bypass mode
		//InputFilter_CI		: 	INT;	// 0: default and will not work (CP defaults to 20ms filter)  7: set filter to less than scan time to be sure to catch all pulses for a chained move
		//SWLimit_Hi_CI		: 	INT;	//software limit switch high (best to make this a retained or persistent variable) mm/deg
		//SWLimit_Lo_CI		: 	INT;	//Software limit switch low (best to make this a retained or persistent variable) mm/deg
		//Limit_NC_NO_CI 		: 	BOOL;	// Using NC limit switches =0; Using NO Limit switches =1; Not suggested to use NO switches		
END_VAR
VAR_OUTPUT
	//Program Outputs
		Out						: LinPPR_Out;
		//Homed_PO				: BOOL;		//true if axis is homed
		//DistancePos_PO			: REAL;		//current position
		//LastDistancePos_PO		: REAL;		//last position
		//ExpDistancePos_PO		: REAL;		//expected position if all pulses are executed
	//Visual outputs (VO)
		//MechTypeMsg_VO			: STRING;	//comment for mech config type
		//ConfigMSG_VO			: STRING;	//comment for config settings
		//ErrorMsg_VO				: STRING;	//message for error description
		//Error2Msg_VO			: STRING;	//second message for error description
		//Error3Msg_VO			: string;	//third message for error description
END_VAR
VAR
	AltSpeedCase		: INT;		//case tracker altspeed()
	AltSpeedReq			: BOOL;		//turn altspeed method on
	HomeCase			: INT;		//case tracker home()
	JogCase				: INT;		//case tracker Jog()
	SuperJogCase		: INT;		//case tracker SuperJog()
	testBOol			: BOOL;		//tester
	error				: INT;		//5: increment error
	PulsesEnabled		: BOOL;		//enable absolute move method to command pulses
	busy				: BOOL;		//move in progress
	MoveComplete		: BOOL;		//all ppr accounted for after move command
	PulseCount			: INT;		//current Pulse Count
	expectedPulse		: INT;		//expected pulses from commanded movements at set PPR
	HomeTrig			: R_trig;	//trigger position capture when homing ends
	ATrig				: R_trig;	//counter/trigger to track how many increments of a output have been commanded
	pulseCounter		: r_trig;
	JogRTrig			: R_Trig;	//jog execute trigger
	JogFTrig			: F_Trig;	//Jog Cancel Trigger
	ASG					: BOOL;		//all systems go clearpath (if using asg)
	Cancelled			: BOOL;		//move was cancelled requires reset
	CW					: BOOL; 	//direction of motor rotation: CW is true;  CCW is false;
	DistanceToGo		: REAL;		//difference in distance from current position and requested position.  used to determine linear direction
	isConfigured		: BOOL;		//turns on or off the configuration settings method so it only runs on first scan
	DistPerMRev 		: INT;
	testlimit			: INT;
	testR				: INT;
	DisPerPulse			: INT;		//distance per pulse based on configuration inputs
	testpulsecnt		: INT;		//testing flot vs int
	PulseQueSet			: BOOL;		//start pulses for move
	PulseQue			: int;		//int counter to hold the number of pulses left to send
	//FI (Field Inputs)

	HLFB_FI	 		AT %I*	: BOOL;		// high level feedback sensors
	bInputBCom_FI	AT %I*	: BOOL;		// check sum for inputb signal	(double check that direction is actually signaled to motor)
	
	//Linear Homing Variables
	bHigh_FI		AT %I*	: BOOL;
	bLow_FI			AT %I*	: BOOL;
	bHome_FI		AT %I*	: BOOL;
	
	//FO (Field Outputs)
	HLFB24V_FO 			AT %Q*	: BOOL :=1;	//high level feedback 24v power if needed to used el2008 //default set to true so that hlfb is fucntional
	EnableOut_FO 		AT %Q* 	: BOOL; 	//enables the clearpath motor
	InputAOut_FO 		AT %Q* 	: BOOL; 	//input A of clearpath motor, output from plc
	InputBOut_FO 		AT %Q* 	: BOOL; 	//input B of clearpath motor, output from plc
	
END_VAR
VAR RETAIN 
	
	
END_VAR

VAR_IN_OUT

END_VAR

(* Checck clearpath settings before use*)
	(* Check the input filter setting for inputA and inputB.   Also check PPR setting, CntsPerPulse, HLFBsetting, and The type of axis,  
		Place clearpath in correct mode of operation Mode for this FB is position 
		Check what Homing setting is used on the clearpath motor	
		check to make sure that the resolution of movement commands matches gearbox compatibiltiy, and plc scan compatability
		
		How the FB works Details:
			1st scan sets configuration using MechDrive_CI()
			Each scan CP motor direction is set based off CW variable
			LocatePosition() drives limit switches and rotary cam limit quadrants
			Pulses are counted using ppr() to move with hlfb rising trig counter.  Expected pulses are tracked with inputA_FO rising trig
			Enable checks for enable signal, cancelled state, and stop_PI state before turning on motor or disenable
			reset: cp motors require an enable off to reset after ac loss...ie estop w/contactor.  it also resets cancelled bit and busy bit (requires reset_vi to run)
			
			Moves are called using homing sequence, Absolute movement, or with manual movement and all require homing.
			after homing absolute movement within software limit_CI is available or manual jog.  Manual jog is set to single pulse method by default
			After Homing Position is tracked using 'DistancePos_PO'
			ABsolute move chains clearpath pulses together to create a smooth motion profile. 
				Pulses sent are tracked against 'DistancePosReq_PI' and 'DistancePos_PO'  When expected pulses are within range of requested position then 'pulsecount' is reset
	*)
(*configruation input setting*)
IF isConfigured = 0 THEN MechDrive_CI();	END_IF	//run once to set configuration on init

//Pin outs Clockwise (CW) or Counter Clockwise (CCW)
IF CW THEN	InputBOut_FO := 1;	ELSE InputBOut_FO := 0; 	END_IF //sets direction of movement at motor - check this (add bcom direction pin check)
LocatePosition();				//rotary position of the cam wheel  //also includes a double sensor check for SensorCheck_PO  //Also locates position for linear system for limit sensors //Limits
//Triggers
	pulseCounter(clk:=HLFB_FI);		//high Level feedback counter based off direction
	HomeTrig(clk:=Out.Homed_PO);		//used in ppr() to set pulses to zero after homing
	ATrig (clk:=InputAOut_FO);		//counts pulses sent to motor (clearpath should move based on InputA Rising Trig (check settings in CP to be sure - options are for rising or falling trig)
	JogRTrig(CLK:=JogExecute_VI);	//Starts Jog()
	JogFTrig(CLK:=JogExecute_VI);	//Cancels Jog() movement
Jog();
SuperJog();
PPR();							//tracking of the Pulses per revolution if using ppr (default for most use cases)
Home();
//moved movedone into movement manula call and abs move call
MoveDone();						//check if movement is complete (will either check pulses against expected pulses or will check for asg
Enable();						//check for motor enable status and try to enable the motor if PowerOn_PI is true
Reset();						//if reset button turn power off, reset cancelled, and reset busy
IF stop_PI THEN CancelMove(); END_IF	//This requires a reset afterwards to move again

METHOD PUBLIC AltSpeed : BOOL
VAR_INPUT
END_VAR
(*clearpath requires at least a 20ms delay where the enable signal is pulsed off to realize alternate speed *)

//start
CASE AltSpeedCase OF
	0:
		altspeedcase :=10;
	10:
		EnableOut_FO :=1 ;
		AltSpeedCase :=20;
	20:
		EnableOut_FO :=1;
		AltSpeedCase :=30;
	30:
		EnableOut_FO := 0 ;
		AltSpeedCase :=40;
	40:
		EnableOut_FO := 0;
		AltSpeedCase := 50;
	50:
		EnableOut_FO := 0 ;
		AltSpeedCase := 60;
	60:	
		EnableOut_FO := 1 ;
		//Look for 'AltSpeedCase' to be set to '0' in the call function
	
	90: //error or message
END_CASE
END_METHOD

METHOD PUBLIC CancelMove : BOOL
VAR_INPUT
END_VAR
EnableOut_FO 	:= 0;		//only way to clear out overstacked increment calls is to turn enable off and then on
//PowerOn_PI		:=0;	//turn off power on [this is a program input and can't be turned off here] check this to see if still needed[was affecting homecase]
Cancelled	:=1;	//cancelled move needs to be reset
expectedpulse := pulsecount;	//resets expected pulse after an estop or limit switch event
Out.DistancePos_PO := Pulsecount/2; //PPRset_CI*1	//resets distance counter to position after a cancelled move
Out.ExpDistancePos_PO := PulseCount/2; //change distancePOs_PO to float if needed
AltSpeedReq :=0;	//clear alt speed mode	
AltSpeedCase :=0;	
InputAOut_FO :=0;
// message (move was canceled)
END_METHOD

METHOD PUBLIC DisToGo : BOOL
VAR_INPUT
END_VAR
IF Out.Homed_PO THEN
	IF DistancePosReq_PI > Out.ExpDistancePos_PO THEN 
		CW := 1;	//move CW to reach req position
	END_IF
	IF DistancePosReq_PI < Out.ExpDistancePos_PO THEN
		CW :=0;	//Move CCW to reach req position
	END_IF
(*	IF PulseQue >0 THEN 
		PulsesEnabled:=1;
		ELSE PulsesEnabled :=0; 
	END_IF *)
	
	IF DistancePosReq_PI = Out.ExpDistancePos_PO THEN 
		PulsesEnabled :=0;
		CW := CW;
		ELSE
			PulsesEnabled := 1;
	END_IF

	ELSE
	//check this (is the homed block required?)
	//Message that Movement cant be made until homing has occured or use manual mode	
	
END_IF

(*
if pulseQue is > 0 then PulseEnabled;
*)
END_METHOD

METHOD PUBLIC Enable : BOOL 	//attempts to enable the motor based on stop_PI, Cancelled, and PowerOn_PI
VAR_INPUT
END_VAR
IF Stop_PI =0 AND cancelled =0 AND PowerOn_PI =1  THEN
	EnableOut_FO :=1;
	IF altSpeedReq THEN
		AltSpeed();				//calls altspeed to cycle thru if homing or manual mode requests a slower mode
	END_IF
	ELSE EnableOut_FO :=0;	//message to say stop is on (check this)
END_IF


//power on

//check if asg

//if no asg power off and repeat
END_METHOD

METHOD PUBLIC Error : BOOL
VAR_INPUT
END_VAR
// if hlfb pulses do not move in set timeframe after movement call then call error for motor
END_METHOD

METHOD PUBLIC Home : BOOL
VAR_INPUT
END_VAR
//limit switch and home switch configuration
IF IN.HomingSet_CI = 2 THEN //homing sensor not used - home to low sensor
bHome_FI := bLow_FI; 
//message homing sensor not used
END_IF
IF IN.HomingSet_CI = 3 THEN //homing sensor not used - home to Hi sensor
	bHome_FI := bHigh_FI; 
	//message homing sensor not used
END_IF
//error catch for if InputBout wire fails and ends up homing unknown direction repeatedly
IF PowerOn_PI = 0 THEN HomeCase :=0; END_IF
IF Stop_PI = 1 THEN HomeCase := 0; END_IF
//check the InputBOut com using EL1008 input channel to determine that the pulse did work
//message
IF bhomestart_PI = 1 THEN HomeCase :=0; AltSpeedReq := 1; AltSpeedCase:=0; END_IF
CASE HomeCase OF
	0://set pulses equal so that movement can begin and check direction
		IF bHomeStart_PI =1 AND Stop_PI = 0  THEN
			HomeCase := 10;
			bhomeStart_PI :=0;
			AltSpeedReq := 1;				//set slow mode and alternate speed in clearpath
			//AltSpeedCase := 0;			//may need this to start slow speed
			ExpectedPulse := PulseCount;	//Make movement available no matter the pulse count discrepancy
			InputAOut_FO :=0;
			Out.Homed_PO :=0;
		END_IF
	(*5:	
		IF Stop_PI = 0  THEN
			HomeCase := 10;
			bhomeStart_PI :=0;
			AltSpeedReq := 1;				//set slow mode and alternate speed in clearpath
			AltSpeedCase := 0;
			ExpectedPulse := PulseCount;	//Make movement available no matter the pulse count discrepancy
			Homed_PO :=0;
		END_IF*)
		
